KUKA KRL program: MyProgram_125().src

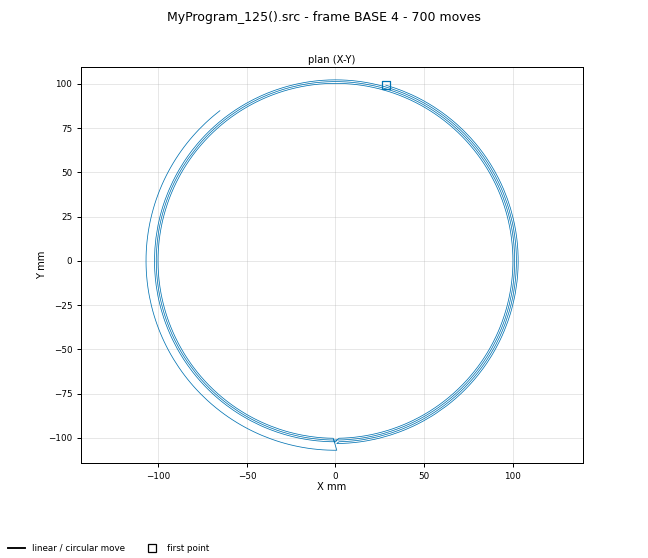
[picture p0: tool path of MyProgram_125().src in frame BASE 4, 700 of 700 moves have a stored position in this frame; points joined in program order, loops and branches not executed]
&ACCESS RVP
&REL 1
&PARAM TEMPLATE = C:\KRC\Roboter\Template\vorgabe
&PARAM EDITMASK = *
DEF MyProgram_125()
; ---- Setting reference (Base) ----
$BASE = BASE_DATA[4]

; --------------------------
; ---- Setting tool (TCP) ----
$TOOL = TOOL_DATA[3]
; --------------------------

$VEL.CP = VEL_APROX_PRINT
Startdeposition()
$VEL.CP = VEL_PRINT
LIN {X 28.4478,Y 99.2015,Z 104,A 68.8345,B 24.9225,C -2.0324,E1 25.0452,E2 376.6609} C_DIS
LIN {X 33.9608,Y 97.4516,Z 104,A 65.4093,B 24.9234,C -2.0215,E1 25.0544,E2 380.1056} C_DIS
LIN {X 37.8064,Y 96.0249,Z 104,A 63.2701,B 24.9231,C -2.0246,E1 25.0599,E2 382.2326} C_DIS
LIN {X 43.2057,Y 93.7204,Z 104,A 59.9493,B 24.9236,C -2.0186,E1 25.0684,E2 385.5597} C_DIS
LIN {X 46.4191,Y 92.1722,Z 104,A 57.9202,B 24.9239,C -2.0142,E1 25.0735,E2 387.5937} C_DIS
LIN {X 49.1956,Y 90.7188,Z 104,A 56.1773,B 24.9241,C -2.0118,E1 25.0778,E2 389.3374} C_DIS
LIN {X 52.6254,Y 88.7733,Z 104,A 54.1134,B 24.924,C -2.0135,E1 25.0828,E2 391.3909} C_DIS
LIN {X 55.7196,Y 86.8644,Z 104,A 52.353,B 24.9234,C -2.0206,E1 25.0869,E2 393.1289} C_DIS
LIN {X 59.6418,Y 84.2205,Z 104,A 49.7177,B 24.9238,C -2.0159,E1 25.093,E2 395.7665} C_DIS
LIN {X 62.8375,Y 81.8632,Z 104,A 47.4109,B 24.9244,C -2.0079,E1 25.0982,E2 398.0838} C_DIS
LIN {X 65.9721,Y 79.3586,Z 104,A 45.1339,B 24.9249,C -2.0018,E1 25.1031,E2 400.3668} C_DIS
LIN {X 68.3933,Y 77.284,Z 104,A 42.4389,B 24.9279,C -1.9615,E1 25.109,E2 403.1461} C_DIS
LIN {X 72.1063,Y 73.8317,Z 104,A 40.6255,B 24.9253,C -1.9955,E1 25.1124,E2 404.8718} C_DIS
LIN {X 76.2514,Y 69.5409,Z 104,A 37.1358,B 24.9264,C -1.9811,E1 25.1192,E2 408.3805} C_DIS
LIN {X 78.8871,Y 66.5371,Z 104,A 34.6809,B 24.9275,C -1.9664,E1 25.1237,E2 410.8588} C_DIS
LIN {X 81.0944,Y 63.8267,Z 104,A 32.6004,B 24.9283,C -1.9561,E1 25.1273,E2 412.9539} C_DIS
LIN {X 83.2071,Y 61.0467,Z 104,A 31.1869,B 24.927,C -1.9726,E1 25.1296,E2 414.3219} C_DIS
LIN {X 85.0597,Y 58.4404,Z 104,A 29.092,B 24.9283,C -1.9551,E1 25.133,E2 416.4478} C_DIS
LIN {X 87.5193,Y 54.6853,Z 104,A 27.0741,B 24.9274,C -1.9679,E1 25.136,E2 418.4253} C_DIS
LIN {X 89.8371,Y 50.7907,Z 104,A 24.5321,B 24.928,C -1.9601,E1 25.1396,E2 420.9726} C_DIS
LIN {X 92.1783,Y 46.4075,Z 104,A 21.5588,B 24.9292,C -1.9436,E1 25.1435,E2 423.9691} C_DIS
LIN {X 93.5017,Y 43.6755,Z 104,A 19.937,B 24.9293,C -1.9415,E1 25.1454,E2 425.5872} C_DIS
LIN {X 95.0517,Y 40.1906,Z 104,A 17.9127,B 24.9295,C -1.9392,E1 25.1476,E2 427.6057} C_DIS
LIN {X 97.219,Y 34.6232,Z 104,A 14.5191,B 24.9304,C -1.9263,E1 25.151,E2 431.011} C_DIS
LIN {X 98.8517,Y 29.6401,Z 104,A 11.6998,B 24.9308,C -1.9213,E1 25.1534,E2 433.826} C_DIS
LIN {X 100.4556,Y 23.6423,Z 104,A 8.2271,B 24.9316,C -1.9096,E1 25.1559,E2 437.3062} C_DIS
LIN {X 101.2146,Y 20.1515,Z 104,A 6.1678,B 24.9323,C -1.9003,E1 25.157,E2 439.3755} C_DIS
LIN {X 101.8875,Y 16.4138,Z 104,A 4.0943,B 24.9327,C -1.8951,E1 25.158,E2 441.4492} C_DIS
LIN {X 102.3864,Y 12.9326,Z 104,A 2.2162,B 24.9329,C -1.892,E1 25.1587,E2 443.3235} C_DIS
LIN {X 102.7618,Y 9.4927,Z 104,A 0.3396,B 24.9332,C -1.8877,E1 25.1592,E2 445.1991} C_DIS
LIN {X 103.034,Y 5.8415,Z 104,A -1.6632,B 24.9336,C -1.8824,E1 25.1596,E2 447.2025} C_DIS
LIN {X 103.1777,Y 2.1249,Z 104,A -3.7158,B 24.934,C -1.8763,E1 25.1598,E2 449.2574} C_DIS
LIN {X 103.1934,Y -1.2746,Z 104,A -5.7366,B 24.9348,C -1.8646,E1 25.1598,E2 451.2936} C_DIS
LIN {X 103.0935,Y -4.6797,Z 104,A -7.9625,B 24.9362,C -1.8447,E1 25.1595,E2 453.5532} C_DIS
LIN {X 102.8699,Y -8.2397,Z 104,A -9.4309,B 24.9352,C -1.8595,E1 25.1592,E2 454.9781} C_DIS
LIN {X 102.5292,Y -11.7444,Z 104,A -11.3324,B 24.9355,C -1.8554,E1 25.1586,E2 456.878} C_DIS
LIN {X 101.5867,Y -18.1732,Z 104,A -15.0021,B 24.9365,C -1.8411,E1 25.1571,E2 460.5598} C_DIS
LIN {X 100.9547,Y -21.415,Z 104,A -17.9326,B 24.9399,C -1.7901,E1 25.1553,E2 463.5936} C_DIS
LIN {X 99.4935,Y -27.4119,Z 104,A -20.2395,B 24.9376,C -1.8252,E1 25.1537,E2 465.8044} C_DIS
LIN {X 98.6543,Y -30.2906,Z 104,A -22.4333,B 24.9394,C -1.7981,E1 25.1519,E2 468.0496} C_DIS
LIN {X 97.4159,Y -34.0627,Z 104,A -23.9606,B 24.938,C -1.8192,E1 25.1505,E2 469.5186} C_DIS
LIN {X 95.3294,Y -39.5318,Z 104,A -27.3157,B 24.939,C -1.8047,E1 25.1471,E2 472.8891} C_DIS
LIN {X 94.0853,Y -42.4035,Z 104,A -29.3837,B 24.9402,C -1.7858,E1 25.1447,E2 474.9904} C_DIS
LIN {X 92.6842,Y -45.3871,Z 104,A -30.6391,B 24.939,C -1.804,E1 25.1433,E2 476.1962} C_DIS
LIN {X 90.0835,Y -50.3494,Z 104,A -33.8809,B 24.94,C -1.7894,E1 25.139,E2 479.4554} C_DIS
LIN {X 88.2478,Y -53.5018,Z 104,A -36.2768,B 24.9414,C -1.7683,E1 25.1355,E2 481.8889} C_DIS
LIN {X 85.5299,Y -57.7474,Z 104,A -38.7285,B 24.941,C -1.7746,E1 25.1318,E2 484.3135} C_DIS
LIN {X 83.4657,Y -60.6935,Z 104,A -40.7287,B 24.9413,C -1.769,E1 25.1285,E2 486.3173} C_DIS
LIN {X 80.5547,Y -64.5089,Z 104,A -43.4191,B 24.9419,C -1.7607,E1 25.1239,E2 489.0144} C_DIS
LIN {X 78.3233,Y -67.199,Z 104,A -45.7003,B 24.9431,C -1.7418,E1 25.1197,E2 491.33} C_DIS
LIN {X 76.0827,Y -69.7246,Z 104,A -47.6961,B 24.9438,C -1.7321,E1 25.1159,E2 493.3398} C_DIS
LIN {X 73.3714,Y -72.5724,Z 104,A -49.2959,B 24.9426,C -1.7504,E1 25.1129,E2 494.8895} C_DIS
LIN {X 70.7262,Y -75.1526,Z 104,A -51.8664,B 24.9443,C -1.7244,E1 25.1076,E2 497.5107} C_DIS
LIN {X 67.9372,Y -77.683,Z 104,A -53.8535,B 24.9443,C -1.7238,E1 25.1034,E2 499.4915} C_DIS
LIN {X 65.3055,Y -79.9092,Z 104,A -55.3491,B 24.9435,C -1.7365,E1 25.1003,E2 500.9515} C_DIS
LIN {X 62.6203,Y -82.0306,Z 104,A -57.2759,B 24.9438,C -1.7313,E1 25.096,E2 502.8835} C_DIS
LIN {X 56.592,Y -86.299,Z 104,A -61.2563,B 24.9441,C -1.7278,E1 25.0869,E2 506.8585} C_DIS
LIN {X 54.3565,Y -87.7246,Z 104,A -63.6703,B 24.9466,C -1.6873,E1 25.081,E2 509.3605} C_DIS
LIN {X 49.7843,Y -90.3991,Z 104,A -65.8005,B 24.9449,C -1.7143,E1 25.076,E2 511.4206} C_DIS
LIN {X 46.4876,Y -92.1374,Z 104,A -67.7484,B 24.9449,C -1.7157,E1 25.0711,E2 513.3598} C_DIS
LIN {X 43.5995,Y -93.5371,Z 104,A -69.6304,B 24.9453,C -1.7089,E1 25.0664,E2 515.253} C_DIS
LIN {X 39.5647,Y -95.3155,Z 104,A -72.0529,B 24.9454,C -1.7062,E1 25.0602,E2 517.676} C_DIS
LIN {X 36.4227,Y -96.5583,Z 104,A -74.8305,B 24.9479,C -1.6682,E1 25.0527,E2 520.5376} C_DIS
LIN {X 31.1049,Y -98.4018,Z 104,A -76.82,B 24.9453,C -1.7089,E1 25.0477,E2 522.427} C_DIS
LIN {X 25.1652,Y -100.0855,Z 104,A -80.3998,B 24.9459,C -1.6992,E1 25.038,E2 526.0241} C_DIS
LIN {X 22.2955,Y -100.7626,Z 104,A -82.8446,B 24.948,C -1.6662,E1 25.0311,E2 528.5437} C_DIS
LIN {X 17.4178,Y -101.7197,Z 104,A -84.8254,B 24.9462,C -1.6942,E1 25.0259,E2 530.456} C_DIS
LIN {X 13.9837,Y -102.249,Z 104,A -86.7797,B 24.9464,C -1.6919,E1 25.0204,E2 532.4141} C_DIS
LIN {X 10.9227,Y -102.6198,Z 104,A -88.4443,B 24.9464,C -1.6927,E1 25.0158,E2 534.0755} C_DIS
LIN {X 7.1827,Y -102.9493,Z 104,A -90.4555,B 24.9462,C -1.6946,E1 25.0102,E2 536.0813} C_DIS
LIN {X 3.9053,Y -103.1268,Z 104,A -92.3624,B 24.9464,C -1.6906,E1 25.0049,E2 537.9971} C_DIS
LIN {X 0.7163,Y -103.1921,Z 104,A -93.4764,B 24.9448,C -1.7156,E1 25.002,E2 539.0514} C_DIS
Enddeposition()
LIN {X 0.7163,Y -103.1921,Z 104,A -93.4764,B 24.9448,C -1.7156,E1 25.002,E2 539.0514} C_DIS
Startdeposition()
$VEL.CP = VEL_PRINT
LIN {X 2.0318,Y -102.1904,Z 104,A -92.5983,B 24.9434,C -1.7384,E1 25.0046,E2 538.1194} C_DIS
LIN {X 5.4073,Y -102.0676,Z 104,A -90.6289,B 24.9431,C -1.7421,E1 25.0101,E2 536.142} C_DIS
LIN {X 8.8529,Y -101.8278,Z 104,A -88.6176,B 24.9429,C -1.7459,E1 25.0157,E2 534.1226} C_DIS
LIN {X 12.4495,Y -101.451,Z 104,A -86.5641,B 24.9427,C -1.7482,E1 25.0214,E2 532.0652} C_DIS
LIN {X 15.9168,Y -100.964,Z 104,A -84.6708,B 24.9428,C -1.7468,E1 25.0266,E2 530.1769} C_DIS
LIN {X 23.8802,Y -99.3823,Z 104,A -80.2486,B 24.9428,C -1.7457,E1 25.0387,E2 525.763} C_DIS
LIN {X 31.2157,Y -97.3275,Z 104,A -76.1945,B 24.9431,C -1.7417,E1 25.0496,E2 521.725} C_DIS
LIN {X 35.7304,Y -95.7631,Z 104,A -73.401,B 24.9426,C -1.7497,E1 25.0569,E2 518.9182} C_DIS
LIN {X 38.3562,Y -94.7408,Z 104,A -71.6056,B 24.9419,C -1.7606,E1 25.0616,E2 517.1011} C_DIS
LIN {X 42.1338,Y -93.1222,Z 104,A -69.5445,B 24.9423,C -1.7543,E1 25.0669,E2 515.0599} C_DIS
LIN {X 44.8643,Y -91.8397,Z 104,A -67.5857,B 24.9414,C -1.7678,E1 25.0719,E2 513.0744} C_DIS
LIN {X 48.1361,Y -90.1678,Z 104,A -65.182,B 24.9403,C -1.7852,E1 25.0779,E2 510.6362} C_DIS
LIN {X 51.0133,Y -88.5699,Z 104,A -63.6781,B 24.941,C -1.7747,E1 25.0815,E2 509.1616} C_DIS
LIN {X 54.2812,Y -86.6057,Z 104,A -61.8626,B 24.9416,C -1.7657,E1 25.0857,E2 507.3731} C_DIS
LIN {X 56.4646,Y -85.1985,Z 104,A -59.6362,B 24.9393,C -1.8,E1 25.0911,E2 505.0731} C_DIS
LIN {X 59.6921,Y -82.9699,Z 104,A -58.2013,B 24.9411,C -1.7733,E1 25.0942,E2 503.7063} C_DIS
LIN {X 61.5117,Y -81.6291,Z 104,A -56.7144,B 24.9403,C -1.7849,E1 25.0976,E2 502.1973} C_DIS
LIN {X 64.3732,Y -79.3919,Z 104,A -54.7579,B 24.9403,C -1.7861,E1 25.1018,E2 500.2452} C_DIS
LIN {X 67.5767,Y -76.685,Z 104,A -52.1982,B 24.9393,C -1.8,E1 25.1073,E2 497.6627} C_DIS
LIN {X 70.1127,Y -74.3721,Z 104,A -50.4933,B 24.9396,C -1.7956,E1 25.1107,E2 495.9752} C_DIS
LIN {X 72.6562,Y -71.8893,Z 104,A -48.5035,B 24.9392,C -1.8003,E1 25.1147,E2 493.9826} C_DIS
LIN {X 75.6848,Y -68.6957,Z 104,A -45.8804,B 24.9384,C -1.813,E1 25.1197,E2 491.3412} C_DIS
LIN {X 78.2611,Y -65.7456,Z 104,A -43.7909,B 24.9384,C -1.8143,E1 25.1235,E2 489.2581} C_DIS
LIN {X 80.4577,Y -63.0375,Z 104,A -41.7397,B 24.9377,C -1.8235,E1 25.1271,E2 487.1947} C_DIS
LIN {X 83.0534,Y -59.575,Z 104,A -39.501,B 24.9377,C -1.8224,E1 25.1307,E2 484.9693} C_DIS
LIN {X 85.0334,Y -56.7151,Z 104,A -37.4787,B 24.9372,C -1.8309,E1 25.1339,E2 482.9371} C_DIS
LIN {X 87.333,Y -53.103,Z 104,A -35.2371,B 24.9372,C -1.8312,E1 25.1372,E2 480.7062} C_DIS
LIN {X 88.9379,Y -50.3728,Z 104,A -32.9579,B 24.9353,C -1.8573,E1 25.1405,E2 478.3771} C_DIS
LIN {X 90.5394,Y -47.4305,Z 104,A -31.3086,B 24.9356,C -1.8533,E1 25.1426,E2 476.7458} C_DIS
LIN {X 92.8479,Y -42.7368,Z 104,A -28.7531,B 24.9361,C -1.8464,E1 25.1456,E2 474.2203} C_DIS
LIN {X 94.1041,Y -39.893,Z 104,A -26.9081,B 24.9354,C -1.856,E1 25.1477,E2 472.3628} C_DIS
LIN {X 95.8184,Y -35.5832,Z 104,A -24.2703,B 24.9348,C -1.8656,E1 25.1504,E2 469.717} C_DIS
LIN {X 98.0268,Y -28.9439,Z 104,A -20.9148,B 24.9355,C -1.8543,E1 25.1533,E2 466.4071} C_DIS
LIN {X 99.1693,Y -24.7532,Z 104,A -17.3798,B 24.9318,C -1.908,E1 25.1558,E2 462.7659} C_DIS
LIN {X 100.0727,Y -20.7966,Z 104,A -15.7776,B 24.9332,C -1.887,E1 25.1567,E2 461.2225} C_DIS
LIN {X 100.6443,Y -17.8267,Z 104,A -13.5604,B 24.9313,C -1.9144,E1 25.1578,E2 458.9539} C_DIS
LIN {X 101.2113,Y -14.2572,Z 104,A -12.1029,B 24.9325,C -1.8971,E1 25.1584,E2 457.5457} C_DIS
LIN {X 101.645,Y -10.737,Z 104,A -10.0993,B 24.932,C -1.9041,E1 25.159,E2 455.5372} C_DIS
LIN {X 101.9598,Y -7.1588,Z 104,A -7.8527,B 24.9309,C -1.9204,E1 25.1595,E2 453.2657} C_DIS
LIN {X 102.1678,Y -2.9603,Z 104,A -5.7845,B 24.9312,C -1.916,E1 25.1597,E2 451.2201} C_DIS
LIN {X 102.209,Y 0.5854,Z 104,A -3.7784,B 24.9307,C -1.9232,E1 25.1597,E2 449.2091} C_DIS
LIN {X 102.128,Y 4.1142,Z 104,A -1.7952,B 24.9302,C -1.9297,E1 25.1596,E2 447.2221} C_DIS
LIN {X 101.9588,Y 7.1745,Z 104,A -0.0066,B 24.9296,C -1.9382,E1 25.1593,E2 445.4243} C_DIS
LIN {X 101.6292,Y 10.8876,Z 104,A 2.0815,B 24.9291,C -1.9448,E1 25.1587,E2 443.333} C_DIS
LIN {X 101.171,Y 14.5409,Z 104,A 4.0601,B 24.9289,C -1.9478,E1 25.158,E2 441.3589} C_DIS
LIN {X 100.5793,Y 18.1877,Z 104,A 6.0958,B 24.9285,C -1.9528,E1 25.157,E2 439.3233} C_DIS
LIN {X 99.8602,Y 21.7929,Z 104,A 8.0959,B 24.9282,C -1.9567,E1 25.1559,E2 437.3256} C_DIS
LIN {X 98.0387,Y 28.9038,Z 104,A 12.7079,B 24.9258,C -1.99,E1 25.1525,E2 432.6617} C_DIS
LIN {X 96.9683,Y 32.3151,Z 104,A 14.5577,B 24.9258,C -1.9895,E1 25.1509,E2 430.8234} C_DIS
LIN {X 94.9077,Y 37.946,Z 104,A 17.6581,B 24.9258,C -1.9886,E1 25.1478,E2 427.7425} C_DIS
LIN {X 93.4849,Y 41.3259,Z 104,A 19.6497,B 24.9256,C -1.9919,E1 25.1456,E2 425.754} C_DIS
LIN {X 92.0858,Y 44.3532,Z 104,A 21.3973,B 24.9256,C -1.9922,E1 25.1435,E2 424.0152} C_DIS
LIN {X 89.9923,Y 48.461,Z 104,A 24.1475,B 24.9245,C -2.0061,E1 25.1399,E2 421.2466} C_DIS
LIN {X 87.3606,Y 53.0577,Z 104,A 26.8354,B 24.9248,C -2.0025,E1 25.1362,E2 418.581} C_DIS
LIN {X 85.9784,Y 55.2693,Z 104,A 28.4265,B 24.9241,C -2.0116,E1 25.1338,E2 416.9764} C_DIS
LIN {X 83.7887,Y 58.5363,Z 104,A 30.7217,B 24.9234,C -2.021,E1 25.1302,E2 414.6706} C_DIS
LIN {X 81.021,Y 62.3105,Z 104,A 32.9926,B 24.924,C -2.0131,E1 25.1264,E2 412.4291} C_DIS
LIN {X 79.3971,Y 64.3668,Z 104,A 34.8502,B 24.9225,C -2.0324,E1 25.1231,E2 410.5346} C_DIS
LIN {X 76.8552,Y 67.3817,Z 104,A 36.9184,B 24.9225,C -2.0317,E1 25.1194,E2 408.4774} C_DIS
LIN {X 72.9414,Y 71.6005,Z 104,A 39.8479,B 24.923,C -2.0268,E1 25.1138,E2 405.5721} C_DIS
LIN {X 70.0401,Y 74.4404,Z 104,A 42.8505,B 24.9204,C -2.0609,E1 25.1076,E2 402.5014} C_DIS
LIN {X 67.4205,Y 76.8214,Z 104,A 44.317,B 24.9217,C -2.044,E1 25.1047,E2 401.0808} C_DIS
LIN {X 65.1003,Y 78.7974,Z 104,A 46.2543,B 24.9207,C -2.0564,E1 25.1005,E2 399.1215} C_DIS
LIN {X 61.6365,Y 81.5354,Z 104,A 48.5805,B 24.9208,C -2.0549,E1 25.0953,E2 396.8074} C_DIS
LIN {X 59.0428,Y 83.4331,Z 104,A 50.5682,B 24.92,C -2.0655,E1 25.0908,E2 394.8017} C_DIS
LIN {X 55.5377,Y 85.8062,Z 104,A 52.689,B 24.9205,C -2.0592,E1 25.0859,E2 392.7026} C_DIS
LIN {X 52.784,Y 87.5269,Z 104,A 54.596,B 24.92,C -2.0654,E1 25.0813,E2 390.7869} C_DIS
LIN {X 49.6591,Y 89.3364,Z 104,A 56.544,B 24.92,C -2.0654,E1 25.0766,E2 388.8451} C_DIS
LIN {X 45.9127,Y 91.32,Z 104,A 58.7528,B 24.9203,C -2.0618,E1 25.0712,E2 386.6507} C_DIS
LIN {X 42.7366,Y 92.848,Z 104,A 61.4103,B 24.918,C -2.091,E1 25.0643,E2 383.9309} C_DIS
LIN {X 39.1814,Y 94.404,Z 104,A 63.1207,B 24.9193,C -2.075,E1 25.06,E2 382.2624} C_DIS
LIN {X 35.8792,Y 95.7067,Z 104,A 65.0437,B 24.9193,C -2.0743,E1 25.055,E2 380.3452} C_DIS
LIN {X 30.0548,Y 97.6921,Z 104,A 68.2912,B 24.9197,C -2.0693,E1 25.0465,E2 377.1157} C_DIS
LIN {X 27.4442,Y 98.4581,Z 104,A 70.0833,B 24.9188,C -2.0807,E1 25.0416,E2 375.2997} C_DIS
LIN {X 23.8209,Y 99.3968,Z 104,A 72.0507,B 24.9191,C -2.0769,E1 25.0363,E2 373.3442} C_DIS
LIN {X 19.9323,Y 100.25,Z 104,A 74.1855,B 24.9193,C -2.0742,E1 25.0305,E2 371.2186} C_DIS
LIN {X 16.9194,Y 100.8004,Z 104,A 75.9542,B 24.9191,C -2.0769,E1 25.0256,E2 369.4454} C_DIS
LIN {X 13.6714,Y 101.2935,Z 104,A 77.9392,B 24.9186,C -2.0828,E1 25.0201,E2 367.4482} C_DIS
LIN {X 10.0554,Y 101.7164,Z 104,A 80.0028,B 24.9186,C -2.084,E1 25.0143,E2 365.3831} C_DIS
LIN {X 6.523,Y 102.0028,Z 104,A 81.8975,B 24.9188,C -2.0806,E1 25.0091,E2 363.4974} C_DIS
LIN {X 3.1443,Y 102.1621,Z 104,A 83.7466,B 24.919,C -2.0787,E1 25.0039,E2 361.6534} C_DIS
LIN {X -0.2843,Y 102.2107,Z 104,A 85.7201,B 24.9188,C -2.0802,E1 24.9984,E2 359.6762} C_DIS
LIN {X -3.7672,Y 102.1429,Z 104,A 87.7501,B 24.9187,C -2.0826,E1 24.9927,E2 357.6404} C_DIS
LIN {X -7.4295,Y 101.9415,Z 104,A 89.795,B 24.9187,C -2.0813,E1 24.987,E2 355.5978} C_DIS
LIN {X -10.8072,Y 101.6377,Z 104,A 91.7223,B 24.9187,C -2.0813,E1 24.9817,E2 353.6694} C_DIS
LIN {X -14.5736,Y 101.1664,Z 104,A 93.6444,B 24.9195,C -2.0724,E1 24.9764,E2 351.7672} C_DIS
LIN {X -17.5168,Y 100.7,Z 104,A 96.2337,B 24.9169,C -2.1054,E1 24.9691,E2 349.0967} C_DIS
LIN {X -22.2225,Y 99.7665,Z 104,A 97.9084,B 24.92,C -2.0653,E1 24.9647,E2 347.5152} C_DIS
LIN {X -26.1409,Y 98.8126,Z 104,A 100.2256,B 24.92,C -2.0652,E1 24.9585,E2 345.1951} C_DIS
LIN {X -29.8055,Y 97.7694,Z 104,A 102.5833,B 24.9196,C -2.071,E1 24.9521,E2 342.8197} C_DIS
LIN {X -34.5878,Y 96.1815,Z 104,A 105.5092,B 24.9196,C -2.0712,E1 24.9443,E2 339.8877} C_DIS
LIN {X -38.4296,Y 94.7109,Z 104,A 107.6812,B 24.9202,C -2.0632,E1 24.9387,E2 337.7301} C_DIS
LIN {X -41.8585,Y 93.2463,Z 104,A 109.7598,B 24.9204,C -2.0597,E1 24.9334,E2 335.6549} C_DIS
LIN {X -46.2039,Y 91.1712,Z 104,A 112.5914,B 24.9204,C -2.0602,E1 24.9263,E2 332.8148} C_DIS
LIN {X -50.3251,Y 88.9645,Z 104,A 115.2237,B 24.9207,C -2.0561,E1 24.9199,E2 330.1847} C_DIS
LIN {X -53.2516,Y 87.2427,Z 104,A 117.5528,B 24.9198,C -2.068,E1 24.9142,E2 327.82} C_DIS
LIN {X -56.4168,Y 85.2301,Z 104,A 119.0691,B 24.9218,C -2.0428,E1 24.9108,E2 326.3588} C_DIS
LIN {X -59.3305,Y 83.2278,Z 104,A 121.6841,B 24.9203,C -2.0615,E1 24.9047,E2 323.6901} C_DIS
LIN {X -62.433,Y 80.9265,Z 104,A 123.3753,B 24.922,C -2.0399,E1 24.9011,E2 322.0443} C_DIS
LIN {X -65.7842,Y 78.229,Z 104,A 125.8181,B 24.9223,C -2.0357,E1 24.8958,E2 319.6023} C_DIS
LIN {X -68.4518,Y 75.9044,Z 104,A 127.7975,B 24.9226,C -2.031,E1 24.8917,E2 317.6261} C_DIS
LIN {X -71.074,Y 73.4541,Z 104,A 129.7879,B 24.9231,C -2.0255,E1 24.8877,E2 315.6406} C_DIS
LIN {X -73.6523,Y 70.8684,Z 104,A 131.7744,B 24.9236,C -2.0184,E1 24.8838,E2 313.6626} C_DIS
LIN {X -76.1152,Y 68.2163,Z 104,A 133.773,B 24.9241,C -2.0122,E1 24.8801,E2 311.6699} C_DIS
LIN {X -78.2146,Y 65.8015,Z 104,A 136.3853,B 24.9222,C -2.0366,E1 24.8752,E2 308.9876} C_DIS
LIN {X -81.0222,Y 62.3084,Z 104,A 138.3699,B 24.9242,C -2.0111,E1 24.8719,E2 307.0541} C_DIS
LIN {X -83.4284,Y 59.0494,Z 104,A 140.9083,B 24.9239,C -2.0144,E1 24.8678,E2 304.4957} C_DIS
LIN {X -85.3541,Y 56.2287,Z 104,A 142.55,B 24.925,C -1.9994,E1 24.8653,E2 302.8814} C_DIS
LIN {X -88.3397,Y 51.414,Z 104,A 145.6585,B 24.9259,C -1.9879,E1 24.8608,E2 299.7844} C_DIS
LIN {X -90.155,Y 48.1605,Z 104,A 148.2456,B 24.9251,C -1.9993,E1 24.8573,E2 297.1565} C_DIS
LIN {X -91.911,Y 44.7169,Z 104,A 149.7435,B 24.9273,C -1.9694,E1 24.8556,E2 295.7217} C_DIS
LIN {X -94.2947,Y 39.4406,Z 104,A 152.5441,B 24.9291,C -1.9441,E1 24.8524,E2 292.9659} C_DIS
LIN {X -96.2542,Y 34.3866,Z 104,A 156.0661,B 24.9286,C -1.9514,E1 24.8488,E2 289.4069} C_DIS
LIN {X -97.2343,Y 31.5036,Z 104,A 157.843,B 24.9288,C -1.9485,E1 24.8473,E2 287.6267} C_DIS
LIN {X -98.1152,Y 28.646,Z 104,A 159.6602,B 24.9288,C -1.9481,E1 24.8458,E2 285.7999} C_DIS
LIN {X -99.0858,Y 25.0825,Z 104,A 161.7417,B 24.9293,C -1.942,E1 24.8443,E2 283.721} C_DIS
LIN {X -100.2284,Y 20.0381,Z 104,A 164.4726,B 24.9304,C -1.9269,E1 24.8427,E2 281.0101} C_DIS
LIN {X -101.3861,Y 12.9563,Z 104,A 168.1157,B 24.9323,C -1.9007,E1 24.8411,E2 277.4077} C_DIS
LIN {X -101.968,Y 7.0375,Z 104,A 171.806,B 24.9322,C -1.9022,E1 24.8401,E2 273.6918} C_DIS
LIN {X -102.2055,Y 1.1281,Z 104,A 175.9132,B 24.931,C -1.919,E1 24.8398,E2 269.5198} C_DIS
LIN {X -102.1747,Y -2.7355,Z 104,A 177.3844,B 24.9332,C -1.8878,E1 24.8398,E2 268.1142} C_DIS
LIN {X -102.057,Y -5.5992,Z 104,A 179.7752,B 24.9316,C -1.91,E1 24.8402,E2 265.6559} C_DIS
LIN {X -101.745,Y -9.7501,Z 104,A -177.8562,B 24.9321,C -1.9038,E1 24.8409,E2 263.2879} C_DIS
LIN {X -101.2561,Y -13.9417,Z 104,A -176.3348,B 24.9347,C -1.8668,E1 24.8414,E2 261.8458} C_DIS
LIN {X -100.3039,Y -19.6526,Z 104,A -172.8275,B 24.9347,C -1.8657,E1 24.8431,E2 258.3203} C_DIS
LIN {X -99.8238,Y -21.9596,Z 104,A -170.9992,B 24.9338,C -1.8794,E1 24.8442,E2 256.4486} C_DIS
LIN {X -98.9574,Y -25.5821,Z 104,A -169.5895,B 24.9359,C -1.8492,E1 24.8451,E2 255.1028} C_DIS
LIN {X -98.3189,Y -27.9353,Z 104,A -168.0818,B 24.9359,C -1.8499,E1 24.8463,E2 253.5845} C_DIS
LIN {X -97.014,Y -32.1795,Z 104,A -165.7195,B 24.9367,C -1.8379,E1 24.8482,E2 251.2371} C_DIS
LIN {X -96.1176,Y -34.763,Z 104,A -163.9646,B 24.9365,C -1.8412,E1 24.8499,E2 249.4646} C_DIS
LIN {X -94.8159,Y -38.1716,Z 104,A -161.2703,B 24.9353,C -1.8582,E1 24.8528,E2 246.7146} C_DIS
LIN {X -93.146,Y -42.081,Z 104,A -159.715,B 24.9378,C -1.8221,E1 24.8544,E2 245.2369} C_DIS
LIN {X -91.9643,Y -44.6059,Z 104,A -156.9636,B 24.9351,C -1.86,E1 24.8579,E2 242.3802} C_DIS
LIN {X -89.3932,Y -49.5575,Z 104,A -154.939,B 24.9385,C -1.812,E1 24.8605,E2 240.4593} C_DIS
LIN {X -87.9312,Y -52.1067,Z 104,A -153.1739,B 24.9385,C -1.8118,E1 24.863,E2 238.6855} C_DIS
LIN {X -85.7229,Y -55.6673,Z 104,A -150.9278,B 24.9391,C -1.802,E1 24.8663,E2 236.4515} C_DIS
LIN {X -83.6764,Y -58.6969,Z 104,A -147.8636,B 24.937,C -1.8333,E1 24.8714,E2 233.2975} C_DIS
LIN {X -80.6176,Y -62.8339,Z 104,A -145.7593,B 24.9394,C -1.7981,E1 24.8748,E2 231.2671} C_DIS
LIN {X -78.4089,Y -65.5677,Z 104,A -143.4122,B 24.9388,C -1.8071,E1 24.879,E2 228.8877} C_DIS
LIN {X -76.1781,Y -68.146,Z 104,A -142.0214,B 24.9403,C -1.784,E1 24.8815,E2 227.5458} C_DIS
LIN {X -74.0229,Y -70.4839,Z 104,A -140.0675,B 24.9402,C -1.7862,E1 24.8853,E2 225.578} C_DIS
LIN {X -71.6417,Y -72.9008,Z 104,A -138.173,B 24.9405,C -1.7819,E1 24.889,E2 223.6857} C_DIS
LIN {X -69.1474,Y -75.2703,Z 104,A -136.3234,B 24.9409,C -1.7752,E1 24.8928,E2 221.8446} C_DIS
LIN {X -66.214,Y -77.8633,Z 104,A -134.3084,B 24.9417,C -1.7644,E1 24.897,E2 219.8474} C_DIS
LIN {X -64.2123,Y -79.5223,Z 104,A -132.5399,B 24.9411,C -1.773,E1 24.9009,E2 218.0518} C_DIS
LIN {X -61.3858,Y -81.7237,Z 104,A -130.6815,B 24.9417,C -1.7639,E1 24.905,E2 216.2082} C_DIS
LIN {X -57.7585,Y -84.3277,Z 104,A -127.6923,B 24.9408,C -1.7776,E1 24.9119,E2 213.1762} C_DIS
LIN {X -55.0501,Y -86.1191,Z 104,A -126.7846,B 24.9432,C -1.7412,E1 24.9138,E2 212.3521} C_DIS
LIN {X -53.0608,Y -87.3586,Z 104,A -124.9799,B 24.9421,C -1.7572,E1 24.9182,E2 210.5037} C_DIS
LIN {X -47.814,Y -90.3374,Z 104,A -121.8972,B 24.9432,C -1.7415,E1 24.9257,E2 207.4494} C_DIS
LIN {X -42.3972,Y -93.0035,Z 104,A -118.3829,B 24.9432,C -1.7421,E1 24.9345,E2 203.9246} C_DIS
LIN {X -40.1098,Y -94.0127,Z 104,A -116.7262,B 24.9426,C -1.7501,E1 24.9388,E2 202.2449} C_DIS
LIN {X -37.0059,Y -95.277,Z 104,A -114.226,B 24.9412,C -1.7717,E1 24.9455,E2 199.688} C_DIS
LIN {X -33.0026,Y -96.7365,Z 104,A -112.7423,B 24.9435,C -1.7355,E1 24.9492,E2 198.2874} C_DIS
LIN {X -28.9921,Y -98.0125,Z 104,A -110.0318,B 24.9428,C -1.747,E1 24.9565,E2 195.5448} C_DIS
LIN {X -25.211,Y -99.0527,Z 104,A -107.7315,B 24.9426,C -1.7496,E1 24.9627,E2 193.2351} C_DIS
LIN {X -20.9459,Y -100.0421,Z 104,A -105.4283,B 24.9431,C -1.7426,E1 24.9689,E2 190.9455} C_DIS
LIN {X -17.5557,Y -100.693,Z 104,A -103.4586,B 24.9431,C -1.7433,E1 24.9744,E2 188.9723} C_DIS
LIN {X -14.1352,Y -101.2286,Z 104,A -101.5457,B 24.9431,C -1.7418,E1 24.9796,E2 187.0613} C_DIS
LIN {X -10.4519,Y -101.6749,Z 104,A -99.4844,B 24.9432,C -1.7408,E1 24.9854,E2 185.001} C_DIS
LIN {X -6.8061,Y -101.9837,Z 104,A -97.4694,B 24.9432,C -1.7394,E1 24.991,E2 182.9886} C_DIS
LIN {X -3.1489,Y -102.162,Z 104,A -95.4548,B 24.9434,C -1.7381,E1 24.9966,E2 180.9765} C_DIS
LIN {X 0.1884,Y -102.2113,Z 104,A -93.4781,B 24.9431,C -1.7426,E1 25.0021,E2 178.9892} C_DIS
LIN {X 0.1884,Y -102.2113,Z 104,A -93.4781,B 24.9431,C -1.7426,E1 25.0021,E2 178.9892} C_DIS
Enddeposition()
LIN {X 0.6899,Y -101.2192,Z 104,A -93.277,B 24.9422,C -1.7567,E1 25.0028,E2 178.7548} C_DIS
Startdeposition()
$VEL.CP = VEL_PRINT
LIN {X -3.1051,Y -101.174,Z 104,A -96.2602,B 24.9443,C -1.7245,E1 24.9943,E2 181.8144} C_DIS
LIN {X -6.2692,Y -101.0288,Z 104,A -98.2117,B 24.9447,C -1.7184,E1 24.9888,E2 183.7808} C_DIS
LIN {X -9.4962,Y -100.7754,Z 104,A -100.0097,B 24.9446,C -1.7198,E1 24.9838,E2 185.5765} C_DIS
LIN {X -13.2088,Y -100.3563,Z 104,A -102.1074,B 24.9446,C -1.7208,E1 24.978,E2 187.6732} C_DIS
LIN {X -16.7473,Y -99.8266,Z 104,A -104.1152,B 24.9444,C -1.722,E1 24.9724,E2 189.6799} C_DIS
LIN {X -20.3984,Y -99.145,Z 104,A -106.1965,B 24.9444,C -1.7236,E1 24.9667,E2 191.7598} C_DIS
LIN {X -26.0843,Y -97.8035,Z 104,A -109.5853,B 24.9444,C -1.7224,E1 24.9575,E2 195.1562} C_DIS
LIN {X -30.1334,Y -96.6324,Z 104,A -111.7792,B 24.9438,C -1.7311,E1 24.9517,E2 197.333} C_DIS
LIN {X -32.984,Y -95.6984,Z 104,A -113.7948,B 24.9445,C -1.7209,E1 24.9463,E2 199.3767} C_DIS
LIN {X -37.1024,Y -94.1766,Z 104,A -116.0253,B 24.9437,C -1.7325,E1 24.9405,E2 201.5843} C_DIS
LIN {X -40.4503,Y -92.7879,Z 104,A -118.0782,B 24.9437,C -1.7346,E1 24.9352,E2 203.637} C_DIS
LIN {X -44.8351,Y -90.7505,Z 104,A -120.8061,B 24.9434,C -1.7381,E1 24.9284,E2 206.3634} C_DIS
LIN {X -47.6742,Y -89.2934,Z 104,A -122.8976,B 24.9439,C -1.7302,E1 24.9231,E2 208.4796} C_DIS
LIN {X -51.5047,Y -87.1383,Z 104,A -125.1295,B 24.9431,C -1.7429,E1 24.9178,E2 210.6878} C_DIS
LIN {X -54.2044,Y -85.4869,Z 104,A -128.3846,B 24.9462,C -1.694,E1 24.9099,E2 214.0697} C_DIS
LIN {X -59.9946,Y -81.5262,Z 104,A -130.8151,B 24.9423,C -1.7548,E1 24.9046,E2 216.3639} C_DIS
LIN {X -62.9212,Y -79.2892,Z 104,A -133.0285,B 24.9423,C -1.754,E1 24.8997,E2 218.5874} C_DIS
LIN {X -65.5848,Y -77.1003,Z 104,A -135.0413,B 24.9423,C -1.7555,E1 24.8954,E2 220.6043} C_DIS
LIN {X -68.3864,Y -74.6265,Z 104,A -137.1323,B 24.9419,C -1.7606,E1 24.891,E2 222.6916} C_DIS
LIN {X -71.0314,Y -72.1137,Z 104,A -139.2117,B 24.9417,C -1.7644,E1 24.8869,E2 224.7706} C_DIS
LIN {X -73.5796,Y -69.5119,Z 104,A -141.2966,B 24.9414,C -1.768,E1 24.8828,E2 226.8557} C_DIS
LIN {X -76.0158,Y -66.8396,Z 104,A -143.4951,B 24.9414,C -1.7673,E1 24.8787,E2 229.0657} C_DIS
LIN {X -78.6676,Y -63.6964,Z 104,A -145.6446,B 24.9407,C -1.779,E1 24.8749,E2 231.1973} C_DIS
LIN {X -83.4744,Y -57.2556,Z 104,A -150.7118,B 24.9411,C -1.7723,E1 24.8665,E2 236.305} C_DIS
LIN {X -85.2936,Y -54.5056,Z 104,A -152.0666,B 24.9396,C -1.7948,E1 24.8645,E2 237.6131} C_DIS
LIN {X -87.1065,Y -51.5585,Z 104,A -154.0646,B 24.9394,C -1.7986,E1 24.8616,E2 239.6123} C_DIS
LIN {X -88.573,Y -48.998,Z 104,A -156.0998,B 24.9399,C -1.7906,E1 24.8588,E2 241.6773} C_DIS
LIN {X -90.7542,Y -44.8276,Z 104,A -158.401,B 24.9386,C -1.8104,E1 24.856,E2 243.9436} C_DIS
LIN {X -92.2312,Y -41.7043,Z 104,A -160.4378,B 24.9384,C -1.8132,E1 24.8536,E2 245.985} C_DIS
LIN {X -94.0103,Y -37.5259,Z 104,A -163.0877,B 24.9381,C -1.8179,E1 24.8507,E2 248.6384} C_DIS
LIN {X -95.3303,Y -34.0332,Z 104,A -165.1999,B 24.9376,C -1.8241,E1 24.8487,E2 250.7476} C_DIS
LIN {X -96.4644,Y -30.6709,Z 104,A -167.0424,B 24.9368,C -1.8358,E1 24.8471,E2 252.5727} C_DIS
LIN {X -97.294,Y -27.925,Z 104,A -168.7674,B 24.9368,C -1.8373,E1 24.8457,E2 254.3042} C_DIS
LIN {X -98.1679,Y -24.6813,Z 104,A -170.8832,B 24.9368,C -1.8358,E1 24.8442,E2 256.4358} C_DIS
LIN {X -99.0004,Y -21.0947,Z 104,A -173.7733,B 24.9382,C -1.8153,E1 24.8425,E2 259.3918} C_DIS
LIN {X -99.9683,Y -15.8848,Z 104,A -175.6235,B 24.9349,C -1.8633,E1 24.8417,E2 261.1386} C_DIS
LIN {X -100.4806,Y -12.229,Z 104,A -178.1218,B 24.9354,C -1.8561,E1 24.8408,E2 263.669} C_DIS
LIN {X -100.94,Y -7.5524,Z 104,A 179.1296,B 24.935,C -1.8616,E1 24.8401,E2 266.4209} C_DIS
LIN {X -101.1419,Y -4.0299,Z 104,A 176.4902,B 24.9361,C -1.8466,E1 24.8398,E2 269.112} C_DIS
LIN {X -101.2175,Y 0.9916,Z 104,A 174.4741,B 24.9335,C -1.8833,E1 24.8398,E2 271.0526} C_DIS
LIN {X -101.0871,Y 5.2285,Z 104,A 172.1293,B 24.9328,C -1.8929,E1 24.8401,E2 273.3887} C_DIS
LIN {X -100.5669,Y 11.4975,Z 104,A 168.5929,B 24.932,C -1.9052,E1 24.841,E2 276.9169} C_DIS
LIN {X -99.8111,Y 16.8399,Z 104,A 165.5415,B 24.9312,C -1.9151,E1 24.8422,E2 279.9629} C_DIS
LIN {X -99.2617,Y 19.8296,Z 104,A 163.4636,B 24.9317,C -1.9086,E1 24.8433,E2 282.0687} C_DIS
LIN {X -98.334,Y 24.005,Z 104,A 161.3169,B 24.9305,C -1.9255,E1 24.8446,E2 284.1875} C_DIS
LIN {X -97.5973,Y 26.8478,Z 104,A 159.498,B 24.9305,C -1.9255,E1 24.846,E2 286.017} C_DIS
LIN {X -96.6189,Y 30.1769,Z 104,A 157.6808,B 24.9297,C -1.9367,E1 24.8474,E2 287.8181} C_DIS
LIN {X -95.5454,Y 33.4202,Z 104,A 155.6337,B 24.9295,C -1.9389,E1 24.8493,E2 289.8717} C_DIS
LIN {X -94.0823,Y 37.3425,Z 104,A 153.404,B 24.9286,C -1.9509,E1 24.8515,E2 292.0853} C_DIS
LIN {X -92.3703,Y 41.3954,Z 104,A 150.7784,B 24.9284,C -1.9539,E1 24.8544,E2 294.7182} C_DIS
LIN {X -90.9986,Y 44.3326,Z 104,A 148.7115,B 24.9286,C -1.9515,E1 24.8569,E2 296.8019} C_DIS
LIN {X -89.489,Y 47.3029,Z 104,A 147.1021,B 24.9275,C -1.9665,E1 24.8589,E2 298.3843} C_DIS
LIN {X -88.1594,Y 49.7386,Z 104,A 145.3666,B 24.9275,C -1.9654,E1 24.8613,E2 300.1314} C_DIS
LIN {X -86.1455,Y 53.1516,Z 104,A 142.1523,B 24.9295,C -1.9392,E1 24.8661,E2 303.4246} C_DIS
LIN {X -83.1146,Y 57.7735,Z 104,A 140.4662,B 24.9253,C -1.9967,E1 24.8686,E2 304.9821} C_DIS
LIN {X -77.5531,Y 65.0504,Z 104,A 134.8769,B 24.9253,C -1.9967,E1 24.8781,E2 310.5982} C_DIS
LIN {X -75.4561,Y 67.47,Z 104,A 133.0241,B 24.925,C -1.9999,E1 24.8815,E2 312.4515} C_DIS
LIN {X -73.0208,Y 70.0986,Z 104,A 130.9821,B 24.9247,C -2.0044,E1 24.8854,E2 314.4915} C_DIS
LIN {X -70.8689,Y 72.2742,Z 104,A 129.1726,B 24.9246,C -2.0059,E1 24.889,E2 316.3051} C_DIS
LIN {X -68.2672,Y 74.7359,Z 104,A 127.1876,B 24.9241,C -2.0122,E1 24.893,E2 318.2834} C_DIS
LIN {X -65.6345,Y 77.058,Z 104,A 124.6058,B 24.9253,C -1.9962,E1 24.8986,E2 320.9132} C_DIS
LIN {X -62.6542,Y 79.5002,Z 104,A 122.2358,B 24.9254,C -1.9944,E1 24.9038,E2 323.2962} C_DIS
LIN {X -59.0243,Y 82.2315,Z 104,A 120.3581,B 24.9232,C -2.0236,E1 24.908,E2 325.1111} C_DIS
LIN {X -55.571,Y 84.6032,Z 104,A 118.0465,B 24.9227,C -2.0303,E1 24.9133,E2 327.4144} C_DIS
LIN {X -53.23,Y 86.0965,Z 104,A 116.3741,B 24.9227,C -2.0298,E1 24.9172,E2 329.0934} C_DIS
LIN {X -50.3268,Y 87.824,Z 104,A 114.5717,B 24.9222,C -2.0371,E1 24.9216,E2 330.8838} C_DIS
LIN {X -47.4693,Y 89.4013,Z 104,A 111.9017,B 24.9241,C -2.0115,E1 24.9283,E2 333.6221} C_DIS
LIN {X -43.3203,Y 91.485,Z 104,A 110.1445,B 24.9215,C -2.0461,E1 24.9325,E2 335.3016} C_DIS
LIN {X -40.0836,Y 92.9477,Z 104,A 108.0762,B 24.9215,C -2.047,E1 24.9378,E2 337.3726} C_DIS
LIN {X -36.9039,Y 94.2546,Z 104,A 106.0697,B 24.9214,C -2.0476,E1 24.943,E2 339.3822} C_DIS
LIN {X -32.7494,Y 95.7783,Z 104,A 103.7591,B 24.9206,C -2.0577,E1 24.949,E2 341.6734} C_DIS
LIN {X -29.099,Y 96.9493,Z 104,A 101.3395,B 24.9211,C -2.0513,E1 24.9555,E2 344.1125} C_DIS
LIN {X -25.6761,Y 97.9122,Z 104,A 99.1387,B 24.9215,C -2.0466,E1 24.9615,E2 346.3278} C_DIS
LIN {X -19.5905,Y 99.3088,Z 104,A 95.6657,B 24.921,C -2.0519,E1 24.971,E2 349.7925} C_DIS
LIN {X -15.2717,Y 100.0631,Z 104,A 92.83,B 24.9219,C -2.041,E1 24.9789,E2 352.6567} C_DIS
LIN {X -11.7332,Y 100.5393,Z 104,A 91.4007,B 24.9202,C -2.0635,E1 24.9827,E2 354.0336} C_DIS
LIN {X -8.6227,Y 100.8552,Z 104,A 89.423,B 24.9207,C -2.0568,E1 24.9882,E2 356.0282} C_DIS
LIN {X -4.9817,Y 101.1008,Z 104,A 87.3682,B 24.9206,C -2.058,E1 24.9939,E2 358.0808} C_DIS
LIN {X -1.3599,Y 101.2137,Z 104,A 85.315,B 24.9206,C -2.0584,E1 24.9997,E2 360.1331} C_DIS
LIN {X 2.1844,Y 101.1986,Z 104,A 83.3234,B 24.9205,C -2.0593,E1 25.0052,E2 362.1224} C_DIS
LIN {X 5.8833,Y 101.0509,Z 104,A 81.2344,B 24.9205,C -2.0596,E1 25.0111,E2 364.21} C_DIS
LIN {X 9.5312,Y 100.7721,Z 104,A 79.3032,B 24.9201,C -2.0646,E1 25.0164,E2 366.1282} C_DIS
LIN {X 13.1692,Y 100.3614,Z 104,A 77.1076,B 24.9205,C -2.0596,E1 25.0225,E2 368.334} C_DIS
LIN {X 16.7947,Y 99.8187,Z 104,A 75.1049,B 24.9203,C -2.0617,E1 25.028,E2 370.3298} C_DIS
LIN {X 22.1583,Y 98.7684,Z 104,A 72.1233,B 24.9201,C -2.0645,E1 25.0362,E2 373.3012} C_DIS
LIN {X 25.1113,Y 98.0574,Z 104,A 70.3014,B 24.9205,C -2.0596,E1 25.0411,E2 375.1319} C_DIS
LIN {X 28.3887,Y 97.16,Z 104,A 68.2809,B 24.9208,C -2.0546,E1 25.0466,E2 377.1609} C_DIS
LIN {X 32.4414,Y 95.8821,Z 104,A 66.0132,B 24.9206,C -2.0579,E1 25.0525,E2 379.4165} C_DIS
LIN {X 35.786,Y 94.6846,Z 104,A 63.9971,B 24.9207,C -2.0559,E1 25.0578,E2 381.4333} C_DIS
LIN {X 38.9287,Y 93.4374,Z 104,A 61.3611,B 24.923,C -2.0265,E1 25.0648,E2 384.1326} C_DIS
LIN {X 42.8431,Y 91.7077,Z 104,A 59.6769,B 24.9211,C -2.0517,E1 25.0689,E2 385.753} C_DIS
LIN {X 46.8166,Y 89.7451,Z 104,A 57.3306,B 24.9208,C -2.0547,E1 25.0747,E2 388.0858} C_DIS
LIN {X 49.5166,Y 88.2834,Z 104,A 55.4673,B 24.9214,C -2.0475,E1 25.0793,E2 389.9607} C_DIS
LIN {X 52.5876,Y 86.4891,Z 104,A 53.4406,B 24.9217,C -2.044,E1 25.0842,E2 391.9894} C_DIS
LIN {X 55.1771,Y 84.8626,Z 104,A 51.5275,B 24.9224,C -2.0342,E1 25.0887,E2 393.9194} C_DIS
LIN {X 58.336,Y 82.7227,Z 104,A 49.3678,B 24.9227,C -2.0306,E1 25.0937,E2 396.0803} C_DIS
LIN {X 61.5273,Y 80.3761,Z 104,A 47.2781,B 24.9225,C -2.0326,E1 25.0983,E2 398.1578} C_DIS
LIN {X 63.9884,Y 78.4309,Z 104,A 45.6639,B 24.9223,C -2.0356,E1 25.1018,E2 399.7589} C_DIS
LIN {X 66.0148,Y 76.734,Z 104,A 43.8094,B 24.9236,C -2.0187,E1 25.1058,E2 401.6462} C_DIS
LIN {X 69.2584,Y 73.818,Z 104,A 41.5674,B 24.9233,C -2.0226,E1 25.1104,E2 403.8699} C_DIS
LIN {X 71.8817,Y 71.2662,Z 104,A 39.5102,B 24.9236,C -2.0187,E1 25.1145,E2 405.9275} C_DIS
LIN {X 74.6368,Y 68.3752,Z 104,A 37.3075,B 24.9238,C -2.016,E1 25.1187,E2 408.127} C_DIS
LIN {X 76.9122,Y 65.8056,Z 104,A 35.2499,B 24.9245,C -2.007,E1 25.1225,E2 410.1966} C_DIS
LIN {X 79.3474,Y 62.8476,Z 104,A 33.1606,B 24.9246,C -2.005,E1 25.1262,E2 412.281} C_DIS
LIN {X 81.6545,Y 59.8194,Z 104,A 31.0339,B 24.9249,C -2.0008,E1 25.1297,E2 414.4075} C_DIS
LIN {X 83.7452,Y 56.8557,Z 104,A 28.9423,B 24.9254,C -1.9941,E1 25.1331,E2 416.5047} C_DIS
LIN {X 85.6296,Y 53.9774,Z 104,A 27.0601,B 24.9256,C -1.9916,E1 25.1359,E2 418.3833} C_DIS
LIN {X 87.4739,Y 50.9359,Z 104,A 24.0044,B 24.9291,C -1.9449,E1 25.1403,E2 421.5334} C_DIS
LIN {X 90.1548,Y 46.021,Z 104,A 21.9181,B 24.9266,C -1.9791,E1 25.1429,E2 423.528} C_DIS
LIN {X 91.9841,Y 42.2494,Z 104,A 19.4212,B 24.9274,C -1.9674,E1 25.1459,E2 426.0391} C_DIS
LIN {X 93.3549,Y 39.1244,Z 104,A 17.5389,B 24.9277,C -1.9638,E1 25.148,E2 427.9195} C_DIS
LIN {X 94.7621,Y 35.5815,Z 104,A 14.9761,B 24.9293,C -1.9412,E1 25.1506,E2 430.5212} C_DIS
LIN {X 95.9468,Y 32.2495,Z 104,A 13.9558,B 24.9269,C -1.9748,E1 25.1514,E2 431.4566} C_DIS
LIN {X 96.7015,Y 29.9105,Z 104,A 12.1027,B 24.9286,C -1.9519,E1 25.153,E2 433.3533} C_DIS
LIN {X 97.712,Y 26.4232,Z 104,A 9.6692,B 24.9301,C -1.9304,E1 25.1549,E2 435.8237} C_DIS
LIN {X 98.5071,Y 23.2904,Z 104,A 8.3962,B 24.9289,C -1.9472,E1 25.1557,E2 437.0496} C_DIS
LIN {X 99.1697,Y 20.2778,Z 104,A 6.5297,B 24.9297,C -1.9369,E1 25.1568,E2 438.9295} C_DIS
LIN {X 99.8234,Y 16.7662,Z 104,A 4.4854,B 24.9302,C -1.9296,E1 25.1578,E2 440.9791} C_DIS
LIN {X 100.3841,Y 12.9943,Z 104,A 2.3828,B 24.9305,C -1.925,E1 25.1586,E2 443.08} C_DIS
LIN {X 100.7797,Y 9.4494,Z 104,A 0.3644,B 24.931,C -1.9186,E1 25.1592,E2 445.1016} C_DIS
LIN {X 101.0469,Y 5.9563,Z 104,A -1.6524,B 24.9315,C -1.9109,E1 25.1596,E2 447.1247} C_DIS
LIN {X 101.1956,Y 2.347,Z 104,A -3.7102,B 24.9321,C -1.9038,E1 25.1598,E2 449.187} C_DIS
LIN {X 101.2165,Y -1.1512,Z 104,A -5.6129,B 24.9323,C -1.9005,E1 25.1598,E2 451.0861} C_DIS
LIN {X 101.1273,Y -4.3689,Z 104,A -7.4876,B 24.9329,C -1.8925,E1 25.1596,E2 452.9685} C_DIS
LIN {X 100.9548,Y -7.3641,Z 104,A -9.2478,B 24.9334,C -1.8844,E1 25.1592,E2 454.7373} C_DIS
LIN {X 100.6055,Y -11.1679,Z 104,A -11.3397,B 24.9337,C -1.8803,E1 25.1586,E2 456.8265} C_DIS
LIN {X 100.1231,Y -14.884,Z 104,A -13.5398,B 24.9344,C -1.8702,E1 25.1578,E2 459.0374} C_DIS
LIN {X 99.5204,Y -18.4891,Z 104,A -15.465,B 24.9344,C -1.8694,E1 25.1569,E2 460.9532} C_DIS
LIN {X 98.1562,Y -24.7266,Z 104,A -18.8369,B 24.9346,C -1.8677,E1 25.1548,E2 464.3096} C_DIS
LIN {X 97.1671,Y -28.365,Z 104,A -21.1947,B 24.9357,C -1.8519,E1 25.153,E2 466.6913} C_DIS
LIN {X 95.6846,Y -33.0234,Z 104,A -23.7237,B 24.9357,C -1.8528,E1 25.1508,E2 469.2036} C_DIS
LIN {X 94.8179,Y -35.4341,Z 104,A -25.4121,B 24.9366,C -1.8387,E1 25.1492,E2 470.9161} C_DIS
LIN {X 93.7607,Y -38.1411,Z 104,A -26.9022,B 24.9366,C -1.8399,E1 25.1476,E2 472.395} C_DIS
LIN {X 92.4131,Y -41.3005,Z 104,A -28.8526,B 24.937,C -1.8337,E1 25.1455,E2 474.3493} C_DIS
LIN {X 91.0345,Y -44.2578,Z 104,A -31.9068,B 24.9406,C -1.7797,E1 25.1416,E2 477.5147} C_DIS
LIN {X 88.1341,Y -49.784,Z 104,A -35.0017,B 24.9402,C -1.7867,E1 25.1374,E2 480.5768} C_DIS
LIN {X 85.7923,Y -53.717,Z 104,A -36.3265,B 24.9372,C -1.8303,E1 25.1357,E2 481.7919} C_DIS
LIN {X 83.838,Y -56.7186,Z 104,A -38.8631,B 24.939,C -1.804,E1 25.1317,E2 484.3781} C_DIS
LIN {X 81.6945,Y -59.7648,Z 104,A -40.9255,B 24.9393,C -1.8,E1 25.1283,E2 486.4399} C_DIS
LIN {X 79.993,Y -62.0244,Z 104,A -42.5217,B 24.9396,C -1.7959,E1 25.1256,E2 488.0382} C_DIS
LIN {X 77.7999,Y -64.7534,Z 104,A -44.4576,B 24.9398,C -1.7925,E1 25.1222,E2 489.9732} C_DIS
LIN {X 75.2848,Y -67.6613,Z 104,A -46.5491,B 24.9399,C -1.7903,E1 25.1184,E2 492.0605} C_DIS
LIN {X 73.7726,Y -69.3067,Z 104,A -47.8859,B 24.9403,C -1.7842,E1 25.1158,E2 493.4057} C_DIS
LIN {X 71.2655,Y -71.8824,Z 104,A -49.9324,B 24.9407,C -1.7787,E1 25.1118,E2 495.4565} C_DIS
LIN {X 68.6329,Y -74.4003,Z 104,A -52.0336,B 24.9411,C -1.7723,E1 25.1075,E2 497.5643} C_DIS
LIN {X 66.3868,Y -76.4113,Z 104,A -53.5657,B 24.9409,C -1.7753,E1 25.1043,E2 499.0833} C_DIS
LIN {X 64.1408,Y -78.3074,Z 104,A -55.3945,B 24.9416,C -1.765,E1 25.1003,E2 500.9294} C_DIS
LIN {X 61.4081,Y -80.4679,Z 104,A -57.4117,B 24.942,C -1.7589,E1 25.0959,E2 502.9535} C_DIS
LIN {X 58.2133,Y -82.8089,Z 104,A -59.6236,B 24.9422,C -1.7554,E1 25.0909,E2 505.1658} C_DIS
LIN {X 55.472,Y -84.6685,Z 104,A -61.3111,B 24.942,C -1.7592,E1 25.087,E2 506.8389} C_DIS
LIN {X 51.2714,Y -87.2762,Z 104,A -64.9786,B 24.9446,C -1.7199,E1 25.078,E2 510.5878} C_DIS
LIN {X 47.152,Y -89.5684,Z 104,A -66.5506,B 24.9421,C -1.7582,E1 25.0744,E2 512.0648} C_DIS
LIN {X 45.3227,Y -90.5088,Z 104,A -68.3224,B 24.9438,C -1.7324,E1 25.0698,E2 513.8928} C_DIS
LIN {X 42.0769,Y -92.0632,Z 104,A -70.1217,B 24.9434,C -1.7384,E1 25.0653,E2 515.6733} C_DIS
LIN {X 38.6495,Y -93.5538,Z 104,A -72.2461,B 24.9436,C -1.735,E1 25.0598,E2 517.8007} C_DIS
LIN {X 35.494,Y -94.7952,Z 104,A -74.2485,B 24.944,C -1.7291,E1 25.0546,E2 519.8126} C_DIS
LIN {X 31.3266,Y -96.2522,Z 104,A -77.1263,B 24.9451,C -1.7115,E1 25.0469,E2 522.7268} C_DIS
LIN {X 27.6088,Y -97.3836,Z 104,A -78.3184,B 24.9427,C -1.7479,E1 25.0439,E2 523.8307} C_DIS
LIN {X 25.3285,Y -98.0015,Z 104,A -80.0808,B 24.9439,C -1.73,E1 25.039,E2 525.6326} C_DIS
LIN {X 22.0269,Y -98.797,Z 104,A -82.6333,B 24.9456,C -1.704,E1 25.0319,E2 528.243} C_DIS
LIN {X 18.0336,Y -99.6023,Z 104,A -84.2362,B 24.944,C -1.729,E1 25.0277,E2 529.7851} C_DIS
LIN {X 15.1112,Y -100.0879,Z 104,A -85.9137,B 24.944,C -1.7277,E1 25.0231,E2 531.4639} C_DIS
LIN {X 11.7517,Y -100.5371,Z 104,A -87.8643,B 24.9442,C -1.7253,E1 25.0177,E2 533.4188} C_DIS
LIN {X 8.1236,Y -100.8951,Z 104,A -89.9046,B 24.9442,C -1.7251,E1 25.012,E2 535.4583} C_DIS
LIN {X 4.5566,Y -101.1192,Z 104,A -92.0208,B 24.9445,C -1.7207,E1 25.0061,E2 537.5841} C_DIS
LIN {X 0.6899,Y -101.2192,Z 104,A -93.2746,B 24.9422,C -1.7556,E1 25.0028,E2 538.7548} C_DIS
Enddeposition()
LIN {X 0.6899,Y -101.2192,Z 104,A -93.2746,B 24.9422,C -1.7556,E1 25.0028,E2 538.7548} C_DIS
Startdeposition()
$VEL.CP = VEL_PRINT
LIN {X 2.0524,Y -100.212,Z 104,A -92.6041,B 24.9414,C -1.7688,E1 25.0047,E2 538.0531} C_DIS
LIN {X 4.9192,Y -100.1139,Z 104,A -91.0207,B 24.9414,C -1.7673,E1 25.0091,E2 536.474} C_DIS
LIN {X 7.9726,Y -99.9152,Z 104,A -89.2684,B 24.9414,C -1.7682,E1 25.014,E2 534.7202} C_DIS
LIN {X 11.038,Y -99.625,Z 104,A -87.3039,B 24.9408,C -1.777,E1 25.0195,E2 532.7362} C_DIS
LIN {X 14.4775,Y -99.1824,Z 104,A -85.5158,B 24.9412,C -1.7709,E1 25.0244,E2 530.9641} C_DIS
LIN {X 17.1346,Y -98.7592,Z 104,A -83.9137,B 24.941,C -1.7745,E1 25.0289,E2 529.355} C_DIS
LIN {X 20.1702,Y -98.1823,Z 104,A -82.1275,B 24.9408,C -1.7768,E1 25.0338,E2 527.5655} C_DIS
LIN {X 23.1653,Y -97.521,Z 104,A -80.2777,B 24.9405,C -1.7822,E1 25.0388,E2 525.7056} C_DIS
LIN {X 26.1201,Y -96.7696,Z 104,A -78.6372,B 24.9406,C -1.7801,E1 25.0432,E2 524.0727} C_DIS
LIN {X 29.6427,Y -95.7492,Z 104,A -76.5372,B 24.9404,C -1.7826,E1 25.0489,E2 521.9703} C_DIS
LIN {X 32.5992,Y -94.7854,Z 104,A -74.6702,B 24.9401,C -1.7883,E1 25.0538,E2 520.0935} C_DIS
LIN {X 35.5088,Y -93.7322,Z 104,A -73.0165,B 24.9402,C -1.7862,E1 25.0581,E2 518.4482} C_DIS
LIN {X 38.3526,Y -92.607,Z 104,A -71.1671,B 24.9398,C -1.7926,E1 25.063,E2 516.5879} C_DIS
LIN {X 41.1766,Y -91.3843,Z 104,A -69.5176,B 24.9398,C -1.791,E1 25.0671,E2 514.9462} C_DIS
LIN {X 43.9883,Y -90.0665,Z 104,A -67.6535,B 24.9394,C -1.7974,E1 25.0719,E2 513.0719} C_DIS
LIN {X 47.2283,Y -88.4106,Z 104,A -65.5777,B 24.9392,C -1.8008,E1 25.077,E2 510.994} C_DIS
LIN {X 50.394,Y -86.6448,Z 104,A -63.5418,B 24.9391,C -1.8031,E1 25.0819,E2 508.9587} C_DIS
LIN {X 53.4207,Y -84.8114,Z 104,A -61.5499,B 24.9389,C -1.8057,E1 25.0867,E2 506.9669} C_DIS
LIN {X 56.2004,Y -82.9947,Z 104,A -59.8098,B 24.9391,C -1.8032,E1 25.0907,E2 505.2386} C_DIS
LIN {X 58.7224,Y -81.2321,Z 104,A -57.8527,B 24.9383,C -1.8146,E1 25.0952,E2 503.2612} C_DIS
LIN {X 61.4198,Y -79.2105,Z 104,A -55.9862,B 24.9382,C -1.8164,E1 25.0993,E2 501.3974} C_DIS
LIN {X 64.0567,Y -77.0931,Z 104,A -54.1132,B 24.938,C -1.8183,E1 25.1034,E2 499.527} C_DIS
LIN {X 66.846,Y -74.6875,Z 104,A -52.0564,B 24.9378,C -1.8212,E1 25.1077,E2 497.4715} C_DIS
LIN {X 69.341,Y -72.3776,Z 104,A -50.0981,B 24.9375,C -1.8264,E1 25.1117,E2 495.5089} C_DIS
LIN {X 71.736,Y -70.0066,Z 104,A -48.0634,B 24.9369,C -1.8354,E1 25.1157,E2 493.4615} C_DIS
LIN {X 74.2582,Y -67.3252,Z 104,A -46.051,B 24.9367,C -1.8371,E1 25.1195,E2 491.4541} C_DIS
LIN {X 76.2983,Y -65.0014,Z 104,A -44.3608,B 24.9367,C -1.8385,E1 25.1226,E2 489.768} C_DIS
LIN {X 78.4418,Y -62.3987,Z 104,A -42.4107,B 24.9362,C -1.8446,E1 25.126,E2 487.8128} C_DIS
LIN {X 80.5079,Y -59.7114,Z 104,A -40.3757,B 24.9356,C -1.8537,E1 25.1294,E2 485.7659} C_DIS
LIN {X 82.298,Y -57.2158,Z 104,A -38.8378,B 24.9359,C -1.8498,E1 25.1319,E2 484.2447} C_DIS
LIN {X 83.6856,Y -55.1664,Z 104,A -37.3271,B 24.9353,C -1.8577,E1 25.1343,E2 482.723} C_DIS
LIN {X 85.6148,Y -52.1222,Z 104,A -35.3592,B 24.9352,C -1.8598,E1 25.1372,E2 480.76} C_DIS
LIN {X 87.2134,Y -49.4045,Z 104,A -33.3856,B 24.9343,C -1.872,E1 25.1399,E2 478.7678} C_DIS
LIN {X 88.9536,Y -46.1973,Z 104,A -31.3177,B 24.9339,C -1.8775,E1 25.1426,E2 476.698} C_DIS
LIN {X 90.6141,Y -42.8493,Z 104,A -29.188,B 24.9335,C -1.8836,E1 25.1452,E2 474.5652} C_DIS
LIN {X 91.8854,Y -40.046,Z 104,A -27.5459,B 24.9335,C -1.8842,E1 25.1471,E2 472.9306} C_DIS
LIN {X 93.2871,Y -36.6623,Z 104,A -25.5663,B 24.9333,C -1.886,E1 25.1491,E2 470.9578} C_DIS
LIN {X 94.1681,Y -34.3362,Z 104,A -24.054,B 24.9327,C -1.8941,E1 25.1506,E2 469.4348} C_DIS
LIN {X 95.3664,Y -30.8521,Z 104,A -21.9576,B 24.9323,C -1.9003,E1 25.1525,E2 467.3356} C_DIS
LIN {X 96.4321,Y -27.3397,Z 104,A -19.9779,B 24.9322,C -1.9021,E1 25.154,E2 465.363} C_DIS
LIN {X 97.2254,Y -24.3759,Z 104,A -18.0302,B 24.9312,C -1.9156,E1 25.1554,E2 463.3947} C_DIS
LIN {X 98.0515,Y -20.8048,Z 104,A -15.9893,B 24.9309,C -1.92,E1 25.1566,E2 461.3551} C_DIS
LIN {X 98.6483,Y -17.7518,Z 104,A -14.3821,B 24.9309,C -1.9188,E1 25.1575,E2 459.7603} C_DIS
LIN {X 99.1511,Y -14.6979,Z 104,A -12.6371,B 24.9306,C -1.9235,E1 25.1582,E2 458.0145} C_DIS
LIN {X 99.5517,Y -11.6648,Z 104,A -10.8948,B 24.9302,C -1.9289,E1 25.1588,E2 456.2697} C_DIS
LIN {X 99.8649,Y -8.6017,Z 104,A -8.941,B 24.9293,C -1.9425,E1 25.1593,E2 454.2954} C_DIS
LIN {X 100.1078,Y -5.029,Z 104,A -7.1086,B 24.9294,C -1.9403,E1 25.1596,E2 452.479} C_DIS
LIN {X 100.2046,Y -2.4518,Z 104,A -5.6559,B 24.9291,C -1.9442,E1 25.1598,E2 451.0258} C_DIS
LIN {X 100.2334,Y 0.2416,Z 104,A -3.9997,B 24.9284,C -1.954,E1 25.1598,E2 449.3564} C_DIS
LIN {X 100.1859,Y 3.0636,Z 104,A -2.4582,B 24.9283,C -1.9562,E1 25.1597,E2 447.8187} C_DIS
LIN {X 100.0223,Y 6.4978,Z 104,A -0.4915,B 24.9278,C -1.9626,E1 25.1594,E2 445.8487} C_DIS
LIN {X 99.807,Y 9.2285,Z 104,A 1.0869,B 24.9274,C -1.9681,E1 25.159,E2 444.2666} C_DIS
LIN {X 99.4031,Y 12.8701,Z 104,A 3.0627,B 24.9272,C -1.97,E1 25.1583,E2 442.2981} C_DIS
LIN {X 98.9697,Y 15.8721,Z 104,A 4.9277,B 24.9264,C -1.9807,E1 25.1575,E2 440.4187} C_DIS
LIN {X 98.4219,Y 18.9668,Z 104,A 6.6734,B 24.9262,C -1.9843,E1 25.1566,E2 438.6748} C_DIS
LIN {X 97.6631,Y 22.5504,Z 104,A 8.6614,B 24.926,C -1.9865,E1 25.1555,E2 436.6931} C_DIS
LIN {X 96.9206,Y 25.5611,Z 104,A 10.407,B 24.9257,C -1.9909,E1 25.1543,E2 434.9474} C_DIS
LIN {X 96.2677,Y 27.9198,Z 104,A 12.0091,B 24.9247,C -2.0034,E1 25.153,E2 433.3249} C_DIS
LIN {X 95.3661,Y 30.8532,Z 104,A 13.6482,B 24.9247,C -2.004,E1 25.1516,E2 431.6936} C_DIS
LIN {X 94.18,Y 34.3036,Z 104,A 15.7374,B 24.9242,C -2.0104,E1 25.1497,E2 429.6011} C_DIS
LIN {X 92.8401,Y 37.78,Z 104,A 17.7359,B 24.9242,C -2.0113,E1 25.1477,E2 427.6115} C_DIS
LIN {X 91.6379,Y 40.6137,Z 104,A 19.6898,B 24.9232,C -2.0242,E1 25.1455,E2 425.6379} C_DIS
LIN {X 90.181,Y 43.7509,Z 104,A 21.4641,B 24.9234,C -2.0216,E1 25.1433,E2 423.8793} C_DIS
LIN {X 88.7128,Y 46.6545,Z 104,A 23.402,B 24.9227,C -2.0299,E1 25.1409,E2 421.9321} C_DIS
LIN {X 87.052,Y 49.6855,Z 104,A 25.3552,B 24.9224,C -2.0344,E1 25.1382,E2 419.9785} C_DIS
LIN {X 85.335,Y 52.5824,Z 104,A 27.3831,B 24.9217,C -2.0436,E1 25.1352,E2 417.9391} C_DIS
LIN {X 83.6892,Y 55.1609,Z 104,A 28.9153,B 24.922,C -2.0395,E1 25.1329,E2 416.4243} C_DIS
LIN {X 81.9575,Y 57.7056,Z 104,A 30.7367,B 24.9215,C -2.0464,E1 25.13,E2 414.5956} C_DIS
LIN {X 80.1406,Y 60.2005,Z 104,A 32.48,B 24.9212,C -2.0499,E1 25.1271,E2 412.8522} C_DIS
LIN {X 78.0673,Y 62.8665,Z 104,A 34.4336,B 24.9208,C -2.0555,E1 25.1238,E2 410.8947} C_DIS
LIN {X 75.8975,Y 65.4717,Z 104,A 36.3907,B 24.9204,C -2.0607,E1 25.1202,E2 408.9341} C_DIS
LIN {X 73.855,Y 67.7646,Z 104,A 38.0771,B 24.9203,C -2.062,E1 25.1171,E2 407.2522} C_DIS
LIN {X 71.5184,Y 70.2269,Z 104,A 40.0626,B 24.9198,C -2.068,E1 25.1132,E2 405.261} C_DIS
LIN {X 69.1198,Y 72.5909,Z 104,A 42.0716,B 24.9192,C -2.0753,E1 25.1091,E2 403.2432} C_DIS
LIN {X 66.41,Y 75.0778,Z 104,A 44.0982,B 24.9192,C -2.0765,E1 25.1049,E2 401.2217} C_DIS
LIN {X 64.0616,Y 77.0891,Z 104,A 45.7783,B 24.9192,C -2.0765,E1 25.1014,E2 399.5482} C_DIS
LIN {X 61.4205,Y 79.21,Z 104,A 47.7372,B 24.9188,C -2.081,E1 25.0971,E2 397.586} C_DIS
LIN {X 58.725,Y 81.2302,Z 104,A 49.6324,B 24.9186,C -2.0832,E1 25.0928,E2 395.6924} C_DIS
LIN {X 56.1975,Y 82.9967,Z 104,A 51.3199,B 24.9186,C -2.0832,E1 25.0889,E2 394.0105} C_DIS
LIN {X 53.6227,Y 84.6852,Z 104,A 53.0686,B 24.9184,C -2.0855,E1 25.0848,E2 392.2622} C_DIS
LIN {X 51.0119,Y 86.2809,Z 104,A 54.8175,B 24.9182,C -2.0882,E1 25.0807,E2 390.5125} C_DIS
LIN {X 48.3386,Y 87.8086,Z 104,A 56.7779,B 24.9174,C -2.0983,E1 25.0758,E2 388.5337} C_DIS
LIN {X 45.594,Y 89.2625,Z 104,A 58.4391,B 24.9176,C -2.0963,E1 25.0717,E2 386.882} C_DIS
LIN {X 42.3007,Y 90.8694,Z 104,A 60.5326,B 24.9174,C -2.0988,E1 25.0665,E2 384.7881} C_DIS
LIN {X 38.9318,Y 92.363,Z 104,A 62.5335,B 24.9175,C -2.097,E1 25.0614,E2 382.7961} C_DIS
LIN {X 36.0771,Y 93.517,Z 104,A 64.2854,B 24.9175,C -2.0985,E1 25.0568,E2 381.0447} C_DIS
LIN {X 33.2052,Y 94.5728,Z 104,A 66.0355,B 24.9173,C -2.1001,E1 25.0522,E2 379.2943} C_DIS
LIN {X 30.2662,Y 95.5559,Z 104,A 68.01,B 24.9166,C -2.1092,E1 25.0469,E2 377.3019} C_DIS
LIN {X 27.3387,Y 96.4324,Z 104,A 69.5476,B 24.9171,C -2.1026,E1 25.0429,E2 375.7827} C_DIS
LIN {X 24.3683,Y 97.2273,Z 104,A 71.4065,B 24.9167,C -2.1075,E1 25.0378,E2 373.9151} C_DIS
LIN {X 21.364,Y 97.9295,Z 104,A 73.1658,B 24.9167,C -2.1082,E1 25.033,E2 372.1564} C_DIS
LIN {X 17.76,Y 98.6468,Z 104,A 75.1623,B 24.9169,C -2.1052,E1 25.0276,E2 370.1694} C_DIS
LIN {X 15.3212,Y 99.0549,Z 104,A 76.5764,B 24.9169,C -2.1057,E1 25.0237,E2 368.7555} C_DIS
LIN {X 12.2716,Y 99.4806,Z 104,A 78.3313,B 24.9169,C -2.1058,E1 25.0188,E2 367.0017} C_DIS
LIN {X 9.2293,Y 99.8069,Z 104,A 80.0848,B 24.9168,C -2.1063,E1 25.0139,E2 365.2483} C_DIS
LIN {X 6.1443,Y 100.0461,Z 104,A 82.0613,B 24.9162,C -2.114,E1 25.0084,E2 363.2544} C_DIS
LIN {X 3.065,Y 100.1859,Z 104,A 83.7153,B 24.9165,C -2.1099,E1 25.0038,E2 361.6105} C_DIS
LIN {X 0.0056,Y 100.2346,Z 104,A 85.5721,B 24.9162,C -2.1135,E1 24.9986,E2 359.7452} C_DIS
LIN {X -3.0535,Y 100.1862,Z 104,A 87.1325,B 24.9168,C -2.1061,E1 24.9943,E2 358.2022} C_DIS
LIN {X -6.1513,Y 100.0457,Z 104,A 89.0963,B 24.9163,C -2.1125,E1 24.9888,E2 356.2228} C_DIS
LIN {X -9.2212,Y 99.8077,Z 104,A 90.7514,B 24.9167,C -2.1078,E1 24.9842,E2 354.5779} C_DIS
LIN {X -12.7863,Y 99.4139,Z 104,A 92.7526,B 24.9169,C -2.1049,E1 24.9787,E2 352.5825} C_DIS
LIN {X -15.9611,Y 98.9555,Z 104,A 94.7322,B 24.9166,C -2.1089,E1 24.9732,E2 350.5916} C_DIS
LIN {X -19.4625,Y 98.3264,Z 104,A 96.731,B 24.9168,C -2.106,E1 24.9677,E2 348.5974} C_DIS
LIN {X -23.0203,Y 97.5546,Z 104,A 98.6696,B 24.9174,C -2.099,E1 24.9624,E2 346.673} C_DIS
LIN {X -26.1322,Y 96.7663,Z 104,A 100.5013,B 24.9175,C -2.0971,E1 24.9575,E2 344.8431} C_DIS
LIN {X -29.0896,Y 95.9207,Z 104,A 102.2596,B 24.9177,C -2.0951,E1 24.9528,E2 343.0866} C_DIS
LIN {X -31.9995,Y 94.9876,Z 104,A 104.1243,B 24.9175,C -2.0973,E1 24.9478,E2 341.2134} C_DIS
LIN {X -35.4306,Y 93.7619,Z 104,A 106.1236,B 24.918,C -2.0916,E1 24.9426,E2 339.2235} C_DIS
LIN {X -38.3585,Y 92.6046,Z 104,A 108.1178,B 24.9176,C -2.096,E1 24.9374,E2 337.2143} C_DIS
LIN {X -41.202,Y 91.3729,Z 104,A 109.7818,B 24.9181,C -2.0896,E1 24.9332,E2 335.5616} C_DIS
LIN {X -44.4703,Y 89.8276,Z 104,A 111.8699,B 24.9183,C -2.0871,E1 24.9279,E2 333.4741} C_DIS
LIN {X -47.2514,Y 88.3985,Z 104,A 113.5492,B 24.9188,C -2.0803,E1 24.9238,E2 331.8064} C_DIS
LIN {X -49.9277,Y 86.9128,Z 104,A 115.4164,B 24.9188,C -2.0814,E1 24.9193,E2 329.9312} C_DIS
LIN {X -53.0755,Y 85.027,Z 104,A 117.5271,B 24.919,C -2.078,E1 24.9142,E2 327.8221} C_DIS
LIN {X -55.7123,Y 83.3252,Z 104,A 119.4199,B 24.919,C -2.078,E1 24.9098,E2 325.9231} C_DIS
LIN {X -58.6884,Y 81.2565,Z 104,A 121.4924,B 24.9194,C -2.0737,E1 24.9051,E2 323.8534} C_DIS
LIN {X -61.5661,Y 79.0978,Z 104,A 123.53,B 24.9197,C -2.0687,E1 24.9006,E2 321.8203} C_DIS
LIN {X -64.2812,Y 76.9066,Z 104,A 125.5675,B 24.92,C -2.0659,E1 24.8962,E2 319.7819} C_DIS
LIN {X -66.8599,Y 74.6751,Z 104,A 127.4328,B 24.9205,C -2.0585,E1 24.8923,E2 317.9267} C_DIS
LIN {X -69.3417,Y 72.3769,Z 104,A 129.3628,B 24.9209,C -2.0538,E1 24.8884,E2 316} C_DIS
LIN {X -71.519,Y 70.2263,Z 104,A 131.1899,B 24.921,C -2.0523,E1 24.8848,E2 314.1689} C_DIS
LIN {X -73.8475,Y 67.7728,Z 104,A 133.04,B 24.9216,C -2.0446,E1 24.8813,E2 312.329} C_DIS
LIN {X -76.097,Y 65.2376,Z 104,A 135.0333,B 24.9218,C -2.0416,E1 24.8776,E2 310.3339} C_DIS
LIN {X -78.2897,Y 62.591,Z 104,A 137.0969,B 24.922,C -2.0398,E1 24.874,E2 308.2649} C_DIS
LIN {X -80.5191,Y 59.6962,Z 104,A 138.9907,B 24.9229,C -2.0275,E1 24.8708,E2 306.3914} C_DIS
LIN {X -82.2907,Y 57.2262,Z 104,A 140.8551,B 24.9229,C -2.0271,E1 24.8678,E2 304.5188} C_DIS
LIN {X -84.3329,Y 54.1716,Z 104,A 142.9681,B 24.9234,C -2.0216,E1 24.8646,E2 302.4082} C_DIS
LIN {X -85.9783,Y 51.5239,Z 104,A 144.6492,B 24.924,C -2.0131,E1 24.8621,E2 300.7389} C_DIS
LIN {X -87.5081,Y 48.8768,Z 104,A 146.4086,B 24.9244,C -2.0084,E1 24.8597,E2 298.9813} C_DIS
LIN {X -88.6783,Y 46.7201,Z 104,A 147.8255,B 24.9246,C -2.0048,E1 24.8578,E2 297.5656} C_DIS
LIN {X -89.8125,Y 44.5007,Z 104,A 149.3584,B 24.9246,C -2.0042,E1 24.8559,E2 296.0258} C_DIS
LIN {X -91.3731,Y 41.2014,Z 104,A 151.4678,B 24.9251,C -1.9988,E1 24.8534,E2 293.9179} C_DIS
LIN {X -92.8258,Y 37.815,Z 104,A 153.4864,B 24.9258,C -1.9894,E1 24.8513,E2 291.9106} C_DIS
LIN {X -93.9589,Y 34.9097,Z 104,A 155.4819,B 24.9257,C -1.9911,E1 24.8493,E2 289.8998} C_DIS
LIN {X -94.9848,Y 32.0078,Z 104,A 157.1474,B 24.9263,C -1.9824,E1 24.8478,E2 288.2454} C_DIS
LIN {X -96.0908,Y 28.5159,Z 104,A 159.1499,B 24.927,C -1.9728,E1 24.8461,E2 286.2545} C_DIS
LIN {X -96.7654,Y 26.1353,Z 104,A 160.6809,B 24.927,C -1.9722,E1 24.845,E2 284.7158} C_DIS
LIN {X -97.5196,Y 23.171,Z 104,A 162.3357,B 24.9277,C -1.9635,E1 24.8439,E2 283.0723} C_DIS
LIN {X -98.0636,Y 20.7484,Z 104,A 163.9749,B 24.9275,C -1.9664,E1 24.8429,E2 281.4164} C_DIS
LIN {X -98.6472,Y 17.7574,Z 104,A 165.5171,B 24.9284,C -1.9541,E1 24.8421,E2 279.8945} C_DIS
LIN {X -99.1459,Y 14.7324,Z 104,A 167.4651,B 24.9284,C -1.955,E1 24.8413,E2 277.9327} C_DIS
LIN {X -99.5505,Y 11.6753,Z 104,A 169.1701,B 24.9289,C -1.9474,E1 24.8407,E2 276.2355} C_DIS
LIN {X -99.9119,Y 8.0137,Z 104,A 171.1832,B 24.9296,C -1.9376,E1 24.8402,E2 274.2338} C_DIS
LIN {X -100.0791,Y 5.5473,Z 104,A 172.5982,B 24.9299,C -1.9331,E1 24.84,E2 272.821} C_DIS
LIN {X -100.2036,Y 2.488,Z 104,A 174.4296,B 24.9302,C -1.9302,E1 24.8398,E2 270.9857} C_DIS
LIN {X -100.233,Y -0.3112,Z 104,A 176.0896,B 24.9304,C -1.927,E1 24.8398,E2 269.323} C_DIS
LIN {X -100.1661,Y -3.7029,Z 104,A 178.1364,B 24.9306,C -1.9244,E1 24.84,E2 267.2702} C_DIS
LIN {X -99.9671,Y -7.3139,Z 104,A -179.797,B 24.931,C -1.9178,E1 24.8403,E2 265.2069} C_DIS
LIN {X -99.6442,Y -10.8539,Z 104,A -177.8891,B 24.9318,C -1.9071,E1 24.8409,E2 263.3131} C_DIS
LIN {X -99.1489,Y -14.7127,Z 104,A -175.4916,B 24.9318,C -1.906,E1 24.8418,E2 260.904} C_DIS
LIN {X -98.5483,Y -18.3076,Z 104,A -173.4072,B 24.9324,C -1.8995,E1 24.8428,E2 258.8227} C_DIS
LIN {X -97.9325,Y -21.3501,Z 104,A -171.8215,B 24.9332,C -1.8876,E1 24.8437,E2 257.2561} C_DIS
LIN {X -97.2522,Y -24.2671,Z 104,A -170.0917,B 24.9335,C -1.8829,E1 24.8448,E2 255.5274} C_DIS
LIN {X -96.6038,Y -26.7339,Z 104,A -168.6286,B 24.9338,C -1.8786,E1 24.8459,E2 254.066} C_DIS
LIN {X -95.7414,Y -29.668,Z 104,A -166.8643,B 24.9342,C -1.8739,E1 24.8473,E2 252.3028} C_DIS
LIN {X -94.8098,Y -32.5268,Z 104,A -165.1332,B 24.9345,C -1.8691,E1 24.8488,E2 250.573} C_DIS
LIN {X -93.9529,Y -34.9261,Z 104,A -163.674,B 24.9348,C -1.8649,E1 24.8502,E2 249.1157} C_DIS
LIN {X -92.8407,Y -37.7785,Z 104,A -161.9023,B 24.9351,C -1.8606,E1 24.8521,E2 247.3443} C_DIS
LIN {X -91.6324,Y -40.6261,Z 104,A -159.9206,B 24.9349,C -1.8628,E1 24.8543,E2 245.3464} C_DIS
LIN {X -90.3423,Y -43.4151,Z 104,A -158.2593,B 24.9355,C -1.8546,E1 24.8563,E2 243.6957} C_DIS
LIN {X -88.69,Y -46.6978,Z 104,A -156.1389,B 24.9359,C -1.8495,E1 24.859,E2 241.5761} C_DIS
LIN {X -86.9099,Y -49.9327,Z 104,A -154.1231,B 24.9365,C -1.8405,E1 24.8617,E2 239.5712} C_DIS
LIN {X -85.3367,Y -52.5797,Z 104,A -152.1442,B 24.9363,C -1.8434,E1 24.8646,E2 237.5752} C_DIS
LIN {X -83.6762,Y -55.1806,Z 104,A -150.4774,B 24.9368,C -1.8355,E1 24.8671,E2 235.9189} C_DIS
LIN {X -81.6099,Y -58.1931,Z 104,A -148.6721,B 24.9379,C -1.8204,E1 24.87,E2 234.1406} C_DIS
LIN {X -80.1741,Y -60.1558,Z 104,A -146.9696,B 24.9374,C -1.8279,E1 24.8728,E2 232.4122} C_DIS
LIN {X -77.9488,Y -63.0128,Z 104,A -144.9686,B 24.9379,C -1.8205,E1 24.8763,E2 230.4193} C_DIS
LIN {X -76.0873,Y -65.249,Z 104,A -143.1728,B 24.9379,C -1.8213,E1 24.8795,E2 228.6134} C_DIS
LIN {X -73.8504,Y -67.7696,Z 104,A -141.2897,B 24.9382,C -1.8155,E1 24.883,E2 226.7358} C_DIS
LIN {X -71.523,Y -70.2222,Z 104,A -139.36,B 24.9385,C -1.8112,E1 24.8868,E2 224.808} C_DIS
LIN {X -69.123,Y -72.5878,Z 104,A -137.3047,B 24.9385,C -1.8117,E1 24.8909,E2 222.7429} C_DIS
LIN {X -66.4639,Y -75.0296,Z 104,A -135.3134,B 24.9389,C -1.805,E1 24.895,E2 220.7595} C_DIS
LIN {X -64.0608,Y -77.0897,Z 104,A -133.5651,B 24.9393,C -1.7994,E1 24.8988,E2 219.0178} C_DIS
LIN {X -61.4053,Y -79.2217,Z 104,A -131.5815,B 24.9395,C -1.7972,E1 24.9031,E2 217.0321} C_DIS
LIN {X -58.7394,Y -81.2196,Z 104,A -129.5631,B 24.9395,C -1.798,E1 24.9077,E2 215.0048} C_DIS
LIN {X -55.7669,Y -83.2882,Z 104,A -127.5062,B 24.9397,C -1.7941,E1 24.9124,E2 212.9501} C_DIS
LIN {X -53.0961,Y -85.0142,Z 104,A -125.7576,B 24.94,C -1.7889,E1 24.9165,E2 211.2085} C_DIS
LIN {X -50.4773,Y -86.5968,Z 104,A -123.8962,B 24.94,C -1.7904,E1 24.921,E2 209.3379} C_DIS
LIN {X -47.7935,Y -88.1044,Z 104,A -122.3448,B 24.9406,C -1.7805,E1 24.9248,E2 207.8055} C_DIS
LIN {X -45.6112,Y -89.2537,Z 104,A -120.8241,B 24.9404,C -1.7827,E1 24.9286,E2 206.2754} C_DIS
LIN {X -42.3141,Y -90.8632,Z 104,A -118.8236,B 24.9408,C -1.7767,E1 24.9336,E2 204.2841} C_DIS
LIN {X -40.0466,Y -91.8851,Z 104,A -117.2966,B 24.9407,C -1.779,E1 24.9375,E2 202.748} C_DIS
LIN {X -36.6611,Y -93.2876,Z 104,A -115.3022,B 24.9411,C -1.7732,E1 24.9426,E2 200.7629} C_DIS
LIN {X -34.3469,Y -94.1642,Z 104,A -113.885,B 24.9411,C -1.772,E1 24.9464,E2 199.3456} C_DIS
LIN {X -32.0137,Y -94.9828,Z 104,A -112.3643,B 24.941,C -1.7748,E1 24.9504,E2 197.8154} C_DIS
LIN {X -28.5257,Y -96.0879,Z 104,A -110.3745,B 24.9413,C -1.7695,E1 24.9557,E2 195.8347} C_DIS
LIN {X -25.979,Y -96.8077,Z 104,A -108.797,B 24.9413,C -1.7709,E1 24.9599,E2 194.2514} C_DIS
LIN {X -22.5869,Y -97.6547,Z 104,A -106.7425,B 24.9412,C -1.7719,E1 24.9655,E2 192.1917} C_DIS
LIN {X -18.9565,Y -98.4239,Z 104,A -104.7343,B 24.9415,C -1.7669,E1 24.971,E2 190.1932} C_DIS
LIN {X -16.5387,Y -98.8589,Z 104,A -103.3292,B 24.9415,C -1.7664,E1 24.9749,E2 188.7877} C_DIS
LIN {X -14.0928,Y -99.2371,Z 104,A -101.8081,B 24.9413,C -1.7701,E1 24.9791,E2 187.2568} C_DIS
LIN {X -10.6379,Y -99.6669,Z 104,A -99.8473,B 24.9413,C -1.7687,E1 24.9845,E2 185.298} C_DIS
LIN {X -7.3711,Y -99.9632,Z 104,A -97.8353,B 24.941,C -1.7737,E1 24.9902,E2 183.273} C_DIS
LIN {X -4.3164,Y -100.1398,Z 104,A -96.2936,B 24.9415,C -1.7661,E1 24.9944,E2 181.7491} C_DIS
LIN {X -1.2386,Y -100.2269,Z 104,A -94.3319,B 24.941,C -1.774,E1 25,E2 179.7686} C_DIS
LIN {X -1.2386,Y -100.2269,Z 104,A -94.3319,B 24.941,C -1.774,E1 25,E2 179.7686} C_DIS
Enddeposition()
LIN {X 0.7445,Y -106.9929,Z 105,A -93.5565,B 24.9489,C -1.6507,E1 25.0013,E2 179.2856} C_DIS
Startdeposition()
$VEL.CP = VEL_PRINT
LIN {X -1.313,Y -106.9894,Z 105,A -94.9358,B 24.9496,C -1.6392,E1 24.9974,E2 180.692} C_DIS
LIN {X -4.5153,Y -106.9002,Z 105,A -96.661,B 24.9496,C -1.6386,E1 24.9926,E2 182.4188} C_DIS
LIN {X -7.2585,Y -106.749,Z 105,A -98.1013,B 24.9496,C -1.6398,E1 24.9885,E2 183.8568} C_DIS
LIN {X -9.7916,Y -106.5465,Z 105,A -99.5524,B 24.9498,C -1.6363,E1 24.9845,E2 185.3169} C_DIS
LIN {X -13.0976,Y -106.1928,Z 105,A -101.264,B 24.9496,C -1.6392,E1 24.9798,E2 187.0226} C_DIS
LIN {X -15.6998,Y -105.8394,Z 105,A -102.671,B 24.9496,C -1.6395,E1 24.9759,E2 188.4301} C_DIS
LIN {X -18.2925,Y -105.4222,Z 105,A -104.078,B 24.9496,C -1.6399,E1 24.972,E2 189.8375} C_DIS
LIN {X -20.8742,Y -104.9415,Z 105,A -105.4855,B 24.9496,C -1.6404,E1 24.9681,E2 191.2454} C_DIS
LIN {X -23.4433,Y -104.3976,Z 105,A -106.8932,B 24.9496,C -1.641,E1 24.9643,E2 192.6535} C_DIS
LIN {X -25.9983,Y -103.7909,Z 105,A -108.3012,B 24.9495,C -1.6417,E1 24.9605,E2 194.0618} C_DIS
LIN {X -28.5376,Y -103.1216,Z 105,A -109.7093,B 24.9495,C -1.6425,E1 24.9567,E2 195.4701} C_DIS
LIN {X -31.0597,Y -102.3902,Z 105,A -111.1176,B 24.9494,C -1.6434,E1 24.9529,E2 196.8787} C_DIS
LIN {X -33.5631,Y -101.5971,Z 105,A -112.7089,B 24.9498,C -1.6372,E1 24.9486,E2 198.4874} C_DIS
LIN {X -36.6233,Y -100.5324,Z 105,A -114.2854,B 24.9493,C -1.645,E1 24.9445,E2 200.0487} C_DIS
LIN {X -39.1584,Y -99.5723,Z 105,A -115.7191,B 24.9492,C -1.647,E1 24.9408,E2 201.4805} C_DIS
LIN {X -41.5121,Y -98.6143,Z 105,A -117.083,B 24.9491,C -1.6483,E1 24.9373,E2 202.8445} C_DIS
LIN {X -43.9197,Y -97.5658,Z 105,A -118.5135,B 24.9491,C -1.6489,E1 24.9336,E2 204.277} C_DIS
LIN {X -46.3009,Y -96.4586,Z 105,A -119.9026,B 24.9489,C -1.6512,E1 24.9301,E2 205.6641} C_DIS
LIN {X -48.6541,Y -95.2932,Z 105,A -121.3125,B 24.9489,C -1.6528,E1 24.9266,E2 207.0739} C_DIS
LIN {X -50.9781,Y -94.0705,Z 105,A -122.723,B 24.9487,C -1.6545,E1 24.9231,E2 208.4844} C_DIS
LIN {X -53.3448,Y -92.7489,Z 105,A -124.1787,B 24.9486,C -1.6564,E1 24.9196,E2 209.9398} C_DIS
LIN {X -55.6049,Y -91.4118,Z 105,A -125.5895,B 24.9485,C -1.6583,E1 24.9162,E2 211.3505} C_DIS
LIN {X -58.1189,Y -89.8352,Z 105,A -127.2071,B 24.9484,C -1.6596,E1 24.9124,E2 212.9701} C_DIS
LIN {X -60.5319,Y -88.229,Z 105,A -128.7416,B 24.9482,C -1.6628,E1 24.9088,E2 214.5021} C_DIS
LIN {X -62.6789,Y -86.7169,Z 105,A -130.1531,B 24.9481,C -1.665,E1 24.9056,E2 215.9134} C_DIS
LIN {X -65.058,Y -84.9446,Z 105,A -131.8503,B 24.9481,C -1.6637,E1 24.9018,E2 217.6197} C_DIS
LIN {X -67.4825,Y -83.0311,Z 105,A -133.4786,B 24.9479,C -1.6677,E1 24.8983,E2 219.2446} C_DIS
LIN {X -69.8878,Y -81.0194,Z 105,A -135.2819,B 24.9479,C -1.6662,E1 24.8944,E2 221.0584} C_DIS
LIN {X -72.3701,Y -78.8074,Z 105,A -136.862,B 24.9473,C -1.6774,E1 24.8912,E2 222.6183} C_DIS
LIN {X -74.2823,Y -77.0076,Z 105,A -138.2957,B 24.9472,C -1.6792,E1 24.8883,E2 224.0535} C_DIS
LIN {X -76.0902,Y -75.2217,Z 105,A -139.7095,B 24.9472,C -1.6801,E1 24.8855,E2 225.4712} C_DIS
LIN {X -78.3921,Y -72.8226,Z 105,A -141.4517,B 24.9468,C -1.6854,E1 24.8822,E2 227.2083} C_DIS
LIN {X -80.1557,Y -70.8768,Z 105,A -142.8647,B 24.9466,C -1.6883,E1 24.8795,E2 228.6207} C_DIS
LIN {X -81.871,Y -68.8883,Z 105,A -144.2781,B 24.9464,C -1.6913,E1 24.877,E2 230.0334} C_DIS
LIN {X -83.5369,Y -66.8584,Z 105,A -145.6917,B 24.9462,C -1.6944,E1 24.8745,E2 231.4463} C_DIS
LIN {X -85.1525,Y -64.7881,Z 105,A -147.1051,B 24.946,C -1.6975,E1 24.8721,E2 232.8589} C_DIS
LIN {X -86.7169,Y -62.6789,Z 105,A -148.6636,B 24.9461,C -1.6953,E1 24.8695,E2 234.4301} C_DIS
LIN {X -88.5733,Y -60.0233,Z 105,A -150.2638,B 24.9455,C -1.7048,E1 24.867,E2 236.0158} C_DIS
LIN {X -90.0654,Y -57.7602,Z 105,A -151.7028,B 24.9453,C -1.709,E1 24.8648,E2 237.452} C_DIS
LIN {X -91.4118,Y -55.6049,Z 105,A -153.1646,B 24.9453,C -1.7088,E1 24.8626,E2 238.9216} C_DIS
LIN {X -93.0971,Y -52.7389,Z 105,A -154.883,B 24.9448,C -1.7159,E1 24.8602,E2 240.6322} C_DIS
LIN {X -94.3633,Y -50.4383,Z 105,A -156.2979,B 24.9446,C -1.7194,E1 24.8583,E2 242.0461} C_DIS
LIN {X -95.5727,Y -48.1073,Z 105,A -157.7126,B 24.9444,C -1.723,E1 24.8565,E2 243.4599} C_DIS
LIN {X -96.7246,Y -45.7473,Z 105,A -159.1275,B 24.9441,C -1.7266,E1 24.8548,E2 244.8738} C_DIS
LIN {X -97.8181,Y -43.3598,Z 105,A -160.5424,B 24.9439,C -1.7303,E1 24.8532,E2 246.2877} C_DIS
LIN {X -98.8528,Y -40.9462,Z 105,A -161.9577,B 24.9436,C -1.7341,E1 24.8517,E2 247.7019} C_DIS
LIN {X -99.8279,Y -38.5079,Z 105,A -163.3729,B 24.9434,C -1.7378,E1 24.8502,E2 249.116} C_DIS
LIN {X -100.7428,Y -36.0464,Z 105,A -164.7883,B 24.9431,C -1.7417,E1 24.8489,E2 250.5303} C_DIS
LIN {X -101.5971,Y -33.5631,Z 105,A -166.2036,B 24.9429,C -1.7455,E1 24.8476,E2 251.9444} C_DIS
LIN {X -102.3902,Y -31.0597,Z 105,A -167.619,B 24.9426,C -1.7494,E1 24.8464,E2 253.3587} C_DIS
LIN {X -103.1517,Y -28.4262,Z 105,A -169.2594,B 24.9428,C -1.7477,E1 24.8452,E2 255.0128} C_DIS
LIN {X -103.9364,Y -25.4016,Z 105,A -170.8023,B 24.9421,C -1.7576,E1 24.8442,E2 256.5411} C_DIS
LIN {X -104.5466,Y -22.7604,Z 105,A -172.2429,B 24.9418,C -1.7625,E1 24.8433,E2 257.9785} C_DIS
LIN {X -105.0568,Y -20.2755,Z 105,A -173.6119,B 24.9415,C -1.7663,E1 24.8425,E2 259.3464} C_DIS
LIN {X -105.5375,Y -17.6032,Z 105,A -175.0747,B 24.9412,C -1.7706,E1 24.8418,E2 260.8077} C_DIS
LIN {X -105.9377,Y -15.0078,Z 105,A -176.5677,B 24.9412,C -1.7719,E1 24.8412,E2 262.3065} C_DIS
LIN {X -106.3455,Y -11.7935,Z 105,A -178.3842,B 24.941,C -1.7744,E1 24.8406,E2 264.1278} C_DIS
LIN {X -106.6586,Y -8.4834,Z 105,A 179.9901,B 24.9402,C -1.7858,E1 24.8402,E2 265.7363} C_DIS
LIN {X -106.8347,Y -5.8633,Z 105,A 178.5533,B 24.94,C -1.7892,E1 24.84,E2 267.1736} C_DIS
LIN {X -106.9464,Y -3.2397,Z 105,A 177.158,B 24.9397,C -1.7941,E1 24.8398,E2 268.5655} C_DIS
LIN {X -106.9944,Y -0.539,Z 105,A 175.6336,B 24.9395,C -1.7959,E1 24.8398,E2 270.0947} C_DIS
LIN {X -106.9652,Y 2.6258,Z 105,A 173.9736,B 24.9391,C -1.8026,E1 24.8398,E2 271.7488} C_DIS
LIN {X -106.8686,Y 5.2501,Z 105,A 172.5573,B 24.9388,C -1.8068,E1 24.84,E2 273.1636} C_DIS
LIN {X -106.7075,Y 7.8712,Z 105,A 171.1411,B 24.9385,C -1.811,E1 24.8403,E2 274.5783} C_DIS
LIN {X -106.4822,Y 10.4876,Z 105,A 169.7253,B 24.9382,C -1.8152,E1 24.8407,E2 275.9926} C_DIS
LIN {X -106.1574,Y 13.3708,Z 105,A 168.0554,B 24.9382,C -1.816,E1 24.8412,E2 277.6705} C_DIS
LIN {X -105.7455,Y 16.3067,Z 105,A 166.5406,B 24.9377,C -1.8238,E1 24.8418,E2 279.1758} C_DIS
LIN {X -105.3135,Y 18.8969,Z 105,A 165.1245,B 24.9374,C -1.828,E1 24.8425,E2 280.5903} C_DIS
LIN {X -104.818,Y 21.4758,Z 105,A 163.7292,B 24.937,C -1.8329,E1 24.8432,E2 281.9822} C_DIS
LIN {X -104.2594,Y 24.0417,Z 105,A 162.3134,B 24.9367,C -1.837,E1 24.8441,E2 283.3965} C_DIS
LIN {X -103.638,Y 26.5931,Z 105,A 160.8764,B 24.9365,C -1.8404,E1 24.8451,E2 284.8338} C_DIS
LIN {X -102.8626,Y 29.4517,Z 105,A 159.2861,B 24.9362,C -1.8452,E1 24.8463,E2 286.4218} C_DIS
LIN {X -102.0013,Y 32.3139,Z 105,A 157.6886,B 24.9358,C -1.8503,E1 24.8476,E2 288.0163} C_DIS
LIN {X -101.1776,Y 34.8074,Z 105,A 156.2729,B 24.9355,C -1.8544,E1 24.8488,E2 289.4304} C_DIS
LIN {X -100.0861,Y 37.826,Z 105,A 154.513,B 24.9353,C -1.8583,E1 24.8505,E2 291.191} C_DIS
LIN {X -99.0843,Y 40.3773,Z 105,A 153.0852,B 24.9349,C -1.8642,E1 24.852,E2 292.6126} C_DIS
LIN {X -97.9534,Y 43.0495,Z 105,A 151.466,B 24.9347,C -1.8666,E1 24.8538,E2 294.2351} C_DIS
LIN {X -96.7246,Y 45.7473,Z 105,A 149.9023,B 24.9343,C -1.8722,E1 24.8556,E2 295.794} C_DIS
LIN {X -95.5727,Y 48.1073,Z 105,A 148.4869,B 24.934,C -1.8761,E1 24.8574,E2 297.2078} C_DIS
LIN {X -94.3633,Y 50.4383,Z 105,A 147.0718,B 24.9338,C -1.8799,E1 24.8592,E2 298.6213} C_DIS
LIN {X -93.0971,Y 52.7389,Z 105,A 145.6563,B 24.9335,C -1.8836,E1 24.8611,E2 300.0352} C_DIS
LIN {X -91.596,Y 55.3019,Z 105,A 143.9542,B 24.9335,C -1.8842,E1 24.8636,E2 301.7448} C_DIS
LIN {X -90.0654,Y 57.7602,Z 105,A 142.4952,B 24.9329,C -1.8919,E1 24.8657,E2 303.1927} C_DIS
LIN {X -88.6208,Y 59.9531,Z 105,A 141.0596,B 24.9327,C -1.8948,E1 24.868,E2 304.6287} C_DIS
LIN {X -87.1228,Y 62.11,Z 105,A 139.6449,B 24.9324,C -1.8984,E1 24.8702,E2 306.0418} C_DIS
LIN {X -85.5214,Y 64.2971,Z 105,A 138.2057,B 24.9321,C -1.9027,E1 24.8726,E2 307.4776} C_DIS
LIN {X -83.9177,Y 66.3765,Z 105,A 136.7912,B 24.9319,C -1.9062,E1 24.8751,E2 308.8905} C_DIS
LIN {X -82.2635,Y 68.416,Z 105,A 135.3769,B 24.9316,C -1.9096,E1 24.8776,E2 310.3033} C_DIS
LIN {X -80.5597,Y 70.4142,Z 105,A 133.9627,B 24.9314,C -1.9129,E1 24.8801,E2 311.716} C_DIS
LIN {X -78.8074,Y 72.3701,Z 105,A 132.5489,B 24.9312,C -1.9162,E1 24.8828,E2 313.1282} C_DIS
LIN {X -77.0076,Y 74.2823,Z 105,A 131.1348,B 24.9309,C -1.9194,E1 24.8855,E2 314.5409} C_DIS
LIN {X -75.1614,Y 76.1498,Z 105,A 129.7422,B 24.9307,C -1.9233,E1 24.8883,E2 315.9301} C_DIS
LIN {X -73.3317,Y 77.9133,Z 105,A 128.3533,B 24.9305,C -1.9255,E1 24.8911,E2 317.3195} C_DIS
LIN {X -71.3975,Y 79.6895,Z 105,A 126.9192,B 24.9303,C -1.9277,E1 24.894,E2 318.7541} C_DIS
LIN {X -69.3558,Y 81.4727,Z 105,A 125.481,B 24.9301,C -1.9315,E1 24.8971,E2 320.1889} C_DIS
LIN {X -67.3355,Y 83.1502,Z 105,A 124.089,B 24.9298,C -1.9351,E1 24.9001,E2 321.5775} C_DIS
LIN {X -65.2746,Y 84.7777,Z 105,A 122.6554,B 24.9297,C -1.9371,E1 24.9032,E2 323.0117} C_DIS
Enddeposition()
END
